Yaskawa INFORM job: X2_100(P)(125,-90).JBI

/JOB
//NAME X2_100(P)(125,-90)
//POS
///NPOS 573,573,573,27,0,0
///TOOL 0
///POSTYPE PULSE
///PULSE
C00000=3858,45070,-46943,-23358,97175,-79306
C00001=-126163,171030,121698,-25332,17066,-72423
///LIMIT ON
C00002=-15532,205449,169164,0,-1122,-37
C00003=-2035,205524,169313,0,-1142,-38
///LIMIT OFF
C00004=-24876,216658,221537,-34735,41227,28422
C00005=-32534,213651,221430,-43713,46730,30831
C00006=-90550,189136,203825,-30202,58765,18284
C00007=-119585,140470,218769,-27614,53519,-2911
C00008=-120519,138494,231532,-24554,52332,-6677
C00009=-121361,123084,224135,-22504,53325,-9347
C00010=-121726,115435,217146,-22627,53645,-9461
C00011=-121876,112275,214159,-22659,53833,-9521
C00012=-121870,108701,209945,-22450,54535,-9681
C00013=-121878,109205,210521,-22481,54446,-9661
C00014=-121910,109175,212145,-22779,53504,-9448
C00015=-121878,109205,210521,-22481,54446,-9661
C00016=-121362,120230,220888,-22358,53819,-9461
C00017=-121399,123144,224213,26030,40987,26163
C00018=-121766,115498,217228,25645,41349,26232
C00019=-121913,110359,211916,25262,41930,26397
C00020=-121910,108768,210034,25105,42240,26494
C00021=-121911,109318,210663,25153,42145,26465
C00022=-121945,109286,212284,25618,41227,26168
C00023=-121911,109318,210663,25153,42145,26465
C00024=-121395,120334,221016,25773,41460,26319
C00025=-121834,122785,223550,29969,46824,26161
C00026=-121859,115436,217233,29902,46923,26193
C00027=-121866,110818,212669,29698,47304,26325
C00028=-121863,108844,210335,29512,47673,26452
C00029=-121935,109447,211025,29521,47579,26410
C00030=-121969,109405,212635,29961,46698,26100
C00031=-121935,109447,211025,29521,47579,26410
C00032=-121897,120013,220389,29693,47285,26314
C00033=-121710,149750,244683,33916,46787,25442
C00034=-122130,167084,227684,35838,62010,28886
C00035=-121679,161325,224182,36290,61247,28722
C00036=-121494,157054,220841,36419,61089,28713
C00037=-121492,155796,219623,36386,61172,28744
C00038=-121498,156274,220057,36390,61156,28737
C00039=-121513,157313,222807,36761,60220,28378
C00040=-121498,156274,220057,36390,61156,28737
C00041=-122131,164491,225278,35793,62131,28930
C00042=-121153,166943,227356,19598,60055,30811
C00043=-121390,161131,223816,19656,59323,30620
C00044=-121486,157179,220857,19658,59138,30564
C00045=-121483,155572,219231,19626,59303,30596
C00046=-121495,156085,219721,19629,59269,30586
C00047=-121510,157133,222481,19854,58176,30378
C00048=-121495,156085,219721,19629,59269,30586
C00049=-121161,164380,224998,19569,60183,30833
C00050=-134270,166899,227330,-30052,67117,-21044
C00051=-134672,161022,223642,-30400,66383,-20931
C00052=-134827,157380,220874,-30511,66205,-20916
C00053=-134816,155436,218995,-30471,66344,-20953
C00054=-134842,155930,219452,-30490,66315,-20951
C00055=-135058,156963,222167,-30845,65285,-20702
C00056=-134842,155930,219452,-30490,66315,-20951
C00057=-134278,164319,224942,-30027,67241,-21080
C00058=-134522,188621,240209,-29351,55882,-39556
C00059=-134281,187845,227413,-27061,47780,-60505
C00060=-134637,183113,225522,-27632,46565,-60252
C00061=-134774,179835,223566,-27858,46107,-60152
C00062=-134763,178280,222255,-27854,46115,-60152
C00063=-134775,178711,222615,-27856,46112,-60156
C00064=-134965,180234,225747,-28400,45052,-59871
C00065=-134775,178711,222615,-27856,46112,-60156
C00066=-134277,185474,225522,-27083,47733,-60488
C00067=-128103,202093,243005,-900,47088,-2105
C00068=-121693,187846,227414,25459,51264,56132
C00069=-121495,183214,225706,25955,50017,55854
C00070=-121414,180043,223882,26152,49543,55743
C00071=-121411,178420,222512,26150,49549,55748
C00072=-121403,178860,222872,26150,49552,55751
C00073=-121416,180408,226053,26590,48508,55442
C00074=-121403,178860,222872,26150,49552,55751
C00075=-121682,185481,225516,25477,51219,56123
C00076=-121689,188183,227953,25513,51119,56094
C00077=-121490,183546,226247,26015,49869,55812
C00078=-121408,180079,224179,26215,49393,55704
C00079=-121407,178755,223064,26213,49397,55705
C00080=-121411,179182,223381,26203,49420,55711
C00081=-121423,180718,226547,26645,48380,55401
C00082=-121411,179182,223381,26203,49420,55711
C00083=-121690,185807,226020,25524,51091,56086
C00084=-123779,190470,236318,58172,45370,-30510
C00085=-122063,184657,229672,57761,45274,-29622
C00086=-121391,180820,225681,57548,45265,-29244
C00087=-121389,179381,224477,57547,45264,-29243
C00088=-121377,179861,224816,57519,45280,-29221
C00089=-121365,178277,221590,56564,45934,-28599
C00090=-121377,179861,224816,57519,45280,-29221
C00091=-121233,179889,223673,56966,45622,-28813
C00092=-120840,179898,223685,57074,45455,-28743
C00093=-121856,179870,223641,56791,45888,-28921
C00094=-124230,188212,233297,57460,45939,-30216
C00095=-135456,214682,237929,8760,44354,-9002
C00096=-135014,207234,230989,8630,44755,-8792
C00097=-134830,202547,226948,8592,44816,-8716
C00098=-134825,201671,226346,8603,44738,-8721
C00099=-134842,202253,226813,8604,44750,-8727
C00100=-134670,200231,223307,8417,45842,-8557
C00101=-134842,202253,226813,8604,44750,-8727
C00102=-135456,212819,236850,8805,44063,-9030
C00103=-144745,210021,243410,8185,41273,-14023
C00104=-162917,179999,233290,6575,38143,-23957
C00105=-161998,172707,226275,6517,38664,-23607
C00106=-162887,167099,219775,6342,39818,-23812
C00107=-162887,165781,218634,6340,39844,-23811
C00108=-162887,166055,218871,6340,39839,-23811
C00109=-162343,164612,215992,6206,40837,-23555
C00110=-162887,166055,218871,6340,39839,-23811
C00111=-162962,177992,231819,6593,38021,-23983
C00112=-147831,180663,236712,-46705,20975,10626
C00113=-148148,173122,227595,-43517,22125,9005
C00114=-148274,168937,222870,-42234,22650,8350
C00115=-148281,167110,221344,-42230,22650,8346
C00116=-148302,167857,221980,-42238,22637,8344
C00117=-147925,166248,218822,-40599,23599,7656
C00118=-148302,167857,221980,-42238,22637,8344
C00119=-147863,178628,235160,-46872,20902,10696
C00120=-134462,161839,227541,-33778,50638,-10353
C00121=-128292,130528,217892,-31335,63768,-21724
C00122=-129684,119449,220047,-34318,57761,-20007
C00123=-130320,112373,214177,-34735,57677,-20053
C00124=-130456,109465,211770,-34840,57652,-20062
C00125=-133214,109388,211257,-36497,57589,-20371
C00126=-136667,109271,210511,-38562,57521,-20784
C00127=-139224,109161,209855,-40060,57485,-21111
C00128=-138850,112080,212320,-39829,57519,-21074
C00129=-138002,119182,218308,-39302,57595,-20992
C00130=-116829,118715,218073,25020,47867,39145
C00131=-117081,112091,213071,24998,47591,39033
C00132=-116945,109370,210997,25124,47467,39017
C00133=-125403,109328,210939,20229,48081,38115
C00134=-125748,112035,212901,19975,48276,38114
C00135=-125224,118667,217955,20186,48522,38233
C00136=-124121,120753,219622,35413,60229,26204
C00137=-123486,114299,214861,35950,59841,26140
C00138=-122342,111487,212696,36731,59624,26198
C00139=-123646,102227,205116,46204,63991,23691
C00140=-125197,104926,207303,45145,64225,23601
C00141=-126541,111461,212474,44185,64527,23570
C00142=-123354,156374,234537,36141,60524,36841
C00143=-123006,163587,222304,33363,70023,40058
C00144=-122562,159556,221336,33872,68682,39742
C00145=-122328,157903,220938,34117,68123,39618
C00146=-120667,157882,220896,34940,67759,39903
C00147=-118950,157779,220838,35793,67346,40185
C00148=-123086,151768,218649,44650,69367,37665
C00149=-123645,153585,219325,44221,69895,37762
C00150=-124560,157673,220588,43425,71117,38069
C00151=-118179,162280,221931,19519,66647,42953
C00152=-118374,158121,220823,19639,65298,42675
C00153=-118267,155527,219476,19766,64809,42612
C00154=-124138,155466,219359,17061,65585,41471
C00155=-124017,158021,220644,17053,66071,41570
C00156=-123705,162202,221801,17023,67409,41838
C00157=-131226,163758,224551,-30632,74582,-25473
C00158=-131671,158900,222412,-31029,73469,-25265
C00159=-131767,156865,221384,-31140,73093,-25182
C00160=-137554,155593,218490,-34050,72807,-26431
C00161=-137282,157641,219617,-33852,73169,-26479
C00162=-136745,162505,221837,-33401,74244,-26683
C00163=-132458,177728,230704,-28826,51363,-58996
C00164=-131589,185090,225420,-26277,57937,-60697
C00165=-131989,181524,225146,-26843,56352,-60401
C00166=-132129,179690,224573,-27052,55792,-60292
C00167=-137018,178141,221655,-27936,55567,-61763
C00168=-136911,179846,222046,-27715,56157,-61897
C00169=-136440,196977,232068,-26852,58624,-62420
C00170=-123981,183157,222393,21512,66418,58052
C00171=-123825,180405,223212,21872,64600,57740
C00172=-123515,178835,223292,22117,63748,57656
C00173=-118554,178759,223273,23717,62772,58838
C00174=-118823,180539,223431,23475,63574,58935
C00175=-119074,183322,222662,23052,65379,59248
C00176=-122702,184077,222510,27150,66928,58165
C00177=-122303,181421,223407,27656,65122,57824
C00178=-121939,179837,223488,27962,64268,57706
C00179=-119147,179825,223466,28889,63614,58349
C00180=-122880,176137,223692,38896,64069,56161
C00181=-123433,177900,223899,38463,64850,56297
C00182=-124245,180658,223301,37680,66520,56676
C00183=-126373,202040,241637,26852,43466,21020
C00184=-128666,178893,235276,24840,16714,-14065
C00185=-128229,171381,226060,22241,18307,-12727
C00186=-128063,167759,221784,21279,19001,-12231
C00187=-126454,168065,222273,20329,18606,-11329
C00188=-113498,168020,221950,9782,17256,-2783
C00189=-116924,165235,218756,37372,21894,-17093
C00190=-117333,168644,222995,38850,21324,-17919
C00191=-117978,176136,232334,42331,20047,-19764
C00192=-122460,189534,236128,2418,24460,-9718
C00193=-126271,180528,223816,-31550,27550,-1309
C00194=-126367,172058,213874,-29849,29054,-2198
C00195=-127090,167664,208219,-28567,29945,-3048
C00196=-142506,160672,196064,-19689,30087,-11601
C00197=-142606,164949,201311,-20262,29094,-11331
C00198=-142831,174249,212461,-21540,27099,-10741
C00199=-90550,189136,203825,-30202,58765,18284
C00200=-32534,213651,221430,-43713,46730,30831
///LIMIT ON
C00201=-2035,205524,169313,0,-1142,-38
///LIMIT OFF
C00202=110357,194361,192639,11084,17793,24068
C00203=114624,170501,213981,27000,30394,20280
C00204=117760,152303,229663,38696,39653,17494
C00205=136745,136971,237540,47053,40245,16937
C00206=146994,113665,215692,48512,45897,19228
C00207=147943,109722,211385,48401,46737,19631
C00208=147915,107740,209041,48089,47029,19824
C00209=147921,108247,209621,48160,46963,19780
C00210=148534,108214,211137,49208,46239,19387
C00211=147921,108247,209621,48160,46963,19780
C00212=146752,119366,220398,48075,46495,19266
C00213=146769,122228,223642,-12245,42312,-23405
C00214=147600,114525,216379,-11673,42843,-23379
C00215=143912,110143,217361,-5106,40312,-21729
C00216=143912,106051,212649,-5023,41107,-21780
C00217=143912,106490,213159,-5032,41020,-21775
C00218=144459,106367,214517,-4806,40132,-21665
C00219=143912,108428,215397,-5071,40640,-21751
C00220=146723,119408,220432,-12150,42825,-23484
C00221=129935,127321,227469,-22947,42372,-25293
C00222=100595,140364,234928,-40781,43967,-29064
C00223=79895,121406,212050,-50395,45854,-33130
C00224=75281,118258,216394,-58069,38031,-30004
C00225=73869,113685,209088,-52247,40421,-30660
C00226=73869,110609,205591,-51722,40783,-30969
C00227=73869,110923,205950,-51776,40745,-30937
C00228=73085,111041,207234,-52885,40146,-30618
C00229=74213,115467,210577,-52057,40483,-30622
C00230=82018,121162,207620,-47441,48027,-34093
C00231=122098,148378,227955,-39779,54040,-25728
C00232=121690,165580,226205,-36203,61926,-29153
C00233=121256,163913,232537,-38022,57992,-27736
C00234=121056,160150,229731,-38195,57784,-27699
C00235=121055,158441,228110,-38151,57879,-27739
C00236=121062,158908,228526,-38154,57867,-27733
C00237=121061,159695,230985,-38583,56988,-27366
C00238=121062,158908,228526,-38154,57867,-27733
C00239=121746,167242,233775,-37439,58860,-27965
C00240=120722,169943,236314,-20799,56253,-30328
C00241=120960,164034,232760,-20897,55487,-30119
C00242=121057,160229,229930,-20909,55300,-30059
C00243=121055,158546,228333,-20881,55408,-30082
C00244=121067,159042,228799,-20882,55381,-30074
C00245=121067,159823,231250,-21156,54345,-29857
C00246=121067,159042,228799,-20882,55381,-30074
C00247=120732,167440,234058,-20772,56349,-30345
C00248=148415,169733,235789,37593,61151,22296
C00249=149007,163695,231894,38120,60456,22164
C00250=149231,159863,228946,38284,60282,22149
C00251=149211,158151,227325,38234,60380,22184
C00252=149239,158627,227750,38254,60361,22183
C00253=149676,159369,230053,38836,59445,21914
C00254=149239,158627,227750,38254,60361,22183
C00255=148408,167213,233502,37553,61243,22331
C00256=120948,174757,250553,37714,32624,49250
C00257=118901,165188,232218,31966,38533,51583
C00258=120946,159930,222884,30547,40745,53182
C00259=121038,156296,220141,30673,40571,53142
C00260=121036,154340,218237,30574,40715,53200
C00261=121048,154616,218515,30593,40687,53192
C00262=121049,155465,220596,31099,39958,52886
C00263=121048,154822,218707,30600,40677,53188
C00264=120729,163160,224069,29968,41598,53447
C00265=121377,165750,226457,-30289,41550,-53313
C00266=121143,159913,222862,-30795,40818,-53099
C00267=121047,156279,220118,-30922,40645,-53059
C00268=121045,154323,218215,-30823,40788,-53119
C00269=121036,154817,218686,-30845,40755,-53109
C00270=121036,155874,221461,-31554,39751,-52691
C00271=121036,154817,218686,-30845,40755,-53109
C00272=121366,163152,224045,-30207,41677,-53367
C00273=121272,196441,225736,-23884,56081,-57724
C00274=121089,199139,236729,-25537,51130,-56524
C00275=121004,196182,235381,-25789,50488,-56375
C00276=121002,194715,234291,-25819,50411,-56355
C00277=121006,195110,234541,-25802,50457,-56365
C00278=121007,196631,237575,-26196,49477,-56088
C00279=121006,195110,234541,-25802,50457,-56365
C00280=121299,201138,236064,-25032,52482,-56815
C00281=121488,201206,234672,-5139,48159,3169
C00282=137298,197580,228407,-4602,50872,8306
C00283=137722,195376,231059,-4778,48135,8578
C00284=139041,199622,244674,-11286,32429,11793
C00285=139041,197484,243237,-11354,32218,11828
C00286=139041,199622,244674,-11286,32429,11793
C00287=138787,198080,241716,-10937,33415,11530
C00288=139041,199622,244674,-11286,32429,11793
C00289=121299,208155,246357,-5458,44546,3313
C00290=123539,200771,239806,-5389,44887,4041
C00291=122594,197682,237757,-5423,44517,3747
C00292=122594,195371,236190,-5443,44297,3759
C00293=122594,197682,237757,-5423,44517,3747
C00294=122571,196051,234778,-5332,45507,3680
C00295=122594,197682,237757,-5423,44517,3747
C00296=121306,206138,245061,-5480,44308,3329
C00297=121658,212256,254439,-6066,40669,6202
C00298=109161,194767,243808,20461,40814,-3758
C00299=110406,186463,235065,20125,41665,-3120
C00300=110426,183388,231339,19860,42333,-2953
C00301=110426,181265,229707,19891,42253,-2973
C00302=110426,182012,230285,19880,42280,-2965
C00303=110530,180795,227899,19582,43058,-2746
C00304=110426,183866,231706,19851,42354,-2947
C00305=142983,174413,229445,40846,25339,-9857
C00306=144224,171221,225776,41394,24787,-9570
C00307=144224,167841,222912,41356,24808,-9552
C00308=144224,168628,223585,41369,24801,-9559
C00309=143936,167289,220827,40018,25660,-8977
C00310=142643,175710,231512,43415,24337,-11034
C00311=138046,186038,246419,52517,22458,-16631
C00312=135775,175505,231782,30106,22895,-7564
C00313=132887,170796,225962,29431,24495,-8118
C00314=133012,167528,222347,28819,24948,-7780
C00315=149327,160096,207563,18098,26717,2120
C00316=142622,177488,230472,24926,23040,-3139
C00317=137477,186722,245503,32144,20066,-8132
C00318=126529,166312,224180,-9540,26920,6556
C00319=130231,155715,216648,-10724,26396,8290
C00320=122698,152468,214837,12997,22490,-4012
C00321=121991,147575,209284,12791,23434,-4123
C00322=141345,142654,200759,11361,23339,4608
C00323=141508,151742,210671,11975,21923,4359
C00324=142241,168295,224091,-11275,28686,12573
C00325=118409,183246,223281,22704,61297,57282
C00326=118581,179790,223172,23116,59682,56982
C00327=119858,177440,221871,23553,59055,57217
C00328=122363,178731,225206,28497,55931,59046
C00329=123595,179764,223148,24469,58676,58234
C00330=123340,183247,223305,24003,60279,58531
C00331=123969,187046,227095,-21794,65540,-58072
C00332=123769,179484,222767,-22062,64364,-57894
C00333=124308,177722,222624,-22031,63705,-57614
C00334=119599,178184,223040,-23554,62794,-58733
C00335=118761,179531,222831,-23662,63378,-59098
C00336=119022,182337,222102,-23232,65173,-59409
C00337=122654,182929,221665,-27319,66777,-58337
C00338=122244,180255,222524,-27832,64982,-57999
C00339=122670,178331,221973,-27828,64506,-57752
C00340=119086,178516,222093,-29014,63676,-58577
C00341=121632,176313,222432,-35609,63813,-57115
C00342=123368,178358,224280,-38654,64701,-56471
C00343=124192,179556,222465,-37876,66329,-56835
C00344=123300,177441,230092,-34884,68799,-44911
C00345=123495,171160,238859,-36432,62561,-41346
C00346=123495,167355,235630,-36422,62587,-41356
C00347=124334,166434,238372,-37436,59393,-39895
C00348=118376,166713,238643,-40516,58128,-40736
C00349=118376,166713,238643,-40516,58128,-40736
C00350=120799,174385,242890,-38781,59689,-40830
C00351=118126,161343,221379,-19792,66498,-43092
C00352=118308,157164,220237,-19921,65161,-42814
C00353=119374,159410,226087,-20289,60239,-41711
C00354=124582,159325,225883,-17950,60958,-40729
C00355=124532,167340,231429,-17858,61624,-40849
C00356=143242,171476,234077,33692,69567,22108
C00357=145029,158578,222871,37922,70344,27214
C00358=146531,156505,221119,38712,69988,27450
C00359=149636,158546,225125,45286,65578,24312
C00360=145593,163818,228591,42995,67071,23935
C00361=129314,152311,241224,32836,60701,20495
C00362=134262,125348,219975,36015,59621,20953
C00363=136200,120757,215933,37173,59474,21178
C00364=138600,121552,220497,48290,55487,21652
C00365=129739,126079,224796,42731,56443,20863
C00366=123968,133718,232687,39402,56414,20088
C00367=116671,118195,219736,-25901,46707,-38928
C00368=118115,111302,212748,-24760,47506,-38978
C00369=118703,106589,208138,-24267,47934,-39019
C00370=126682,106493,207892,-19649,48585,-38165
C00371=117444,111276,212730,-25153,47452,-39048
C00372=124109,119988,219209,-35802,60097,-26259
C00373=123452,113507,214395,-36349,59725,-26200
C00374=123794,109050,210148,-36021,60020,-26273
C00375=117612,109054,210103,-40010,59333,-26782
C00376=118160,111552,216388,-45062,55465,-25714
C00377=121329,120470,223550,-42877,55942,-25575
C00378=129083,121917,227984,-46752,58292,-19813
C00379=114229,133215,224760,-34569,55636,-15897
C00380=115215,137513,213650,-31198,63454,-18326
C00381=115698,129470,194907,-29425,69976,-20075
C00382=106762,152299,200628,-28970,57173,-24551
C00383=106762,152299,184780,-28970,-3668,-24551
C00384=106762,172700,182835,-23749,-4416,-26879
C00385=106762,173596,155880,-23749,-4416,-26879
C00386=27327,173596,155880,-23749,-4416,-26879
C00387=61821,209309,227101,13653,32656,17858
C00388=117760,152303,229663,38696,39653,17494
C00389=136745,136971,237540,47053,40245,16937
C00390=146994,113665,215692,48512,45897,19228
C00391=147943,109722,211385,48401,46737,19631
C00392=147915,107740,209041,48089,47029,19824
C00393=147921,108247,209621,48160,46963,19780
C00394=148534,108214,211137,49208,46239,19387
C00395=147921,108247,209621,48160,46963,19780
C00396=146752,119366,220398,48075,46495,19266
C00397=146769,122228,223642,-12245,42312,-23405
C00398=147600,114525,216379,-11673,42843,-23379
C00399=150410,110151,217690,-10757,39930,-22674
C00400=147891,107738,209025,-11299,43871,-23478
C00401=153573,108674,222079,-9620,36586,-21959
C00402=148504,108258,211178,-11182,42854,-23269
C00403=153573,108674,222079,-9620,36586,-21959
C00404=146723,119408,220432,-12150,42825,-23484
C00405=129935,127321,227469,-22947,42372,-25293
C00406=100595,140364,234928,-40781,43967,-29064
C00407=81913,119649,206036,-47366,48141,-34193
C00408=81142,111914,198932,-47506,48252,-34466
C00409=80567,105530,192695,-47437,48513,-34785
C00410=80567,103424,190213,-47154,48820,-34981
C00411=79896,104610,192938,-48190,47941,-34592
C00412=79367,104896,194278,-48926,47369,-34348
C00413=81288,108115,194243,-46832,48931,-34860
C00414=82018,116513,202458,-46931,48572,-34441
C00415=122104,148543,228477,-39885,53858,-25643
C00416=121690,165580,226205,-36203,61926,-29153
C00417=121228,159785,222619,-36652,61188,-29000
C00418=121039,155988,219702,-36787,61016,-28984
C00419=121038,154211,217971,-36739,61139,-29031
C00420=121044,154693,218413,-36744,61121,-29023
C00421=121043,155760,221200,-37127,60178,-28661
C00422=121044,154693,218413,-36744,61121,-29023
C00423=121694,162967,223761,-36153,62058,-29201
C00424=120722,165761,226456,-19970,59936,-31049
C00425=120948,159926,222866,-20032,59223,-30862
C00426=121040,156088,219926,-20029,59083,-30814
C00427=121038,154338,218222,-19999,59222,-30841
C00428=121049,154854,218719,-20002,59186,-30831
C00429=121049,155913,221496,-20240,58090,-30621
C00430=121049,154854,218719,-20002,59186,-30831
C00431=120732,163185,224070,-19939,60073,-31072
C00432=147021,165785,226508,35831,64459,23179
C00433=147568,159794,222565,36267,63796,23080
C00434=147776,155921,219507,36395,63658,23083
C00435=147758,154144,217781,36345,63784,23124
C00436=147784,154635,218233,36365,63757,23122
C00437=148179,155632,220846,36870,62776,22859
C00438=147784,154635,218233,36365,63757,23122
C00439=147016,163193,224095,35787,64586,23223
C00440=120935,171934,242189,34504,35645,50983
C00441=120720,165768,226479,30046,41476,53396
C00442=120946,159930,222884,30547,40745,53182
C00443=121038,156296,220141,30673,40571,53142
C00444=121036,154340,218237,30574,40715,53200
C00445=121048,154616,218515,30593,40687,53192
C00446=121049,155465,220596,31099,39958,52886
C00447=121048,154822,218707,30600,40677,53188
C00448=120729,163160,224069,29968,41598,53447
C00449=121377,165750,226457,-30289,41550,-53313
C00450=121143,159913,222862,-30795,40818,-53099
C00451=121047,156279,220118,-30922,40645,-53059
C00452=121045,154323,218215,-30823,40788,-53119
C00453=121036,154817,218686,-30845,40755,-53109
C00454=121036,155874,221461,-31554,39751,-52691
C00455=121036,154817,218686,-30845,40755,-53109
C00456=121366,163152,224045,-30207,41677,-53367
C00457=121272,196441,225736,-23884,56081,-57724
C00458=121073,192434,224897,-24336,54621,-57437
C00459=120992,189535,223518,-24533,54018,-57314
C00460=120990,188039,222350,-24548,53971,-57303
C00461=120994,188436,222615,-24536,54010,-57311
C00462=120994,190244,226010,-24889,52951,-57041
C00463=120994,188436,222615,-24536,54010,-57311
C00464=121274,194182,224023,-23912,55983,-57699
C00465=121488,201206,234672,-5139,48159,3169
C00466=137298,197580,228407,-4602,50872,8306
C00467=137298,191509,224279,-4639,50294,8333
C00468=139269,198483,245774,-16664,26320,14172
C00469=139269,196637,244517,-16766,26152,14223
C00470=139269,198483,245774,-16664,26320,14172
C00471=139075,197379,243601,-16166,27033,13866
C00472=139269,198483,245774,-16664,26320,14172
C00473=121273,201949,235341,-5146,48120,3100
C00474=123414,194344,228329,-5073,48626,3789
C00475=122511,191235,226161,-5095,48321,3503
C00476=122511,188904,224500,-5108,48148,3511
C00477=122511,191235,226161,-5095,48321,3503
C00478=122490,189334,222835,-5015,49386,3440
C00479=122511,191235,226161,-5095,48321,3503
C00480=121280,199935,233985,-5161,47920,3112
C00481=121614,206656,244155,-5683,44100,5953
C00482=121602,191150,235422,-5966,40449,9428
C00483=121174,183490,227904,-5875,41115,9232
C00484=121005,180342,224725,-5833,41444,9150
C00485=121003,177643,222663,-5847,41326,9158
C00486=121008,178404,223350,-5851,41294,9161
C00487=121008,176471,219820,-5719,42467,9082
C00488=121008,178404,223350,-5851,41294,9161
C00489=121606,189290,234231,-5993,40228,9445
C00490=147345,179625,236056,47140,21312,-11138
C00491=147690,172068,226895,43950,22458,-9504
C00492=147826,168050,222291,42659,22984,-8839
C00493=147834,166033,220594,42645,22988,-8830
C00494=147855,166783,221239,42657,22973,-8830
C00495=147492,165159,218049,41004,23935,-8131
C00496=147855,166783,221239,42657,22973,-8830
C00497=147377,177583,234490,47295,21243,-11203
C00498=135775,175505,231782,30106,22895,-7564
C00499=139825,168083,220832,25470,24638,-4146
C00500=139700,165046,217320,24964,25206,-3934
C00501=152174,156983,201769,15688,28186,4094
C00502=150364,166319,215167,18488,25143,2197
C00503=147525,184400,240334,25395,19839,-1947
C00504=126529,166312,224180,-9540,26920,6556
C00505=130231,155715,216648,-10724,26396,8290
C00506=130045,149819,208548,-10003,28305,7869
C00507=131869,147843,216891,-25172,12050,11560
C00508=149055,140634,197724,-21214,26307,18683
C00509=148313,150562,204331,-12308,32779,14754
C00510=148313,166205,218654,-12570,32021,14892
C00511=118409,183246,223281,22704,61297,57282
C00512=118581,179790,223172,23116,59682,56982
C00513=119613,177433,221860,23486,59108,57157
C00514=124091,177390,221715,24682,58266,58283
C00515=123595,179764,223148,24469,58676,58234
C00516=123340,183247,223305,24003,60279,58531
C00517=123938,190075,227776,-21625,66593,-58285
C00518=123769,179484,222767,-22062,64364,-57894
C00519=123980,177747,222673,-22141,63629,-57689
C00520=118975,177987,223072,-23779,62559,-58856
C00521=118761,179531,222831,-23662,63378,-59098
C00522=119022,182337,222102,-23232,65173,-59409
C00523=122654,182929,221665,-27319,66777,-58337
C00524=122244,180255,222524,-27832,64982,-57999
C00525=122348,178243,222080,-27959,64333,-57799
C00526=119084,177910,221892,-29058,63509,-58532
C00527=123183,174594,222305,-38836,64062,-56290
C00528=123368,176775,223017,-38664,64673,-56460
C00529=124192,179556,222465,-37876,66329,-56835
C00530=123300,177441,230092,-34884,68799,-44911
C00531=122965,162591,221617,-33646,69855,-40187
C00532=122509,158537,220602,-34164,68528,-39873
C00533=122656,156640,219931,-34208,68093,-39694
C00534=118888,156854,220084,-36079,67235,-40332
C00535=123197,150890,218022,-44883,69229,-37756
C00536=123579,152565,218570,-44547,69710,-37880
C00537=124509,156681,219892,-43743,70915,-38181
C00538=118126,161343,221379,-19792,66498,-43092
C00539=118308,157164,220237,-19921,65161,-42814
C00540=119071,154535,218903,-19652,64761,-42579
C00541=124368,154518,218802,-17210,65477,-41554
C00542=123968,157132,220198,-17330,65894,-41703
C00543=123666,161333,221389,-17292,67221,-41971
C00544=144355,163571,225284,37353,71372,27423
C00545=145029,158578,222871,37922,70344,27214
C00546=146175,156230,221157,38559,69945,27345
C00547=151129,153949,216102,40712,70190,28712
C00548=150395,156248,217650,40288,70560,28668
C00549=149652,161243,220185,39700,71542,28858
C00550=132795,148549,237387,35039,60818,21489
C00551=129694,120788,221943,34103,57517,19821
C00552=131382,111553,213551,35044,57698,20084
C00553=143552,107861,207554,42137,57676,21682
C00554=150345,107155,204350,45732,57861,22855
C00555=138916,111308,211941,39557,57554,20977
C00556=138073,118434,217968,39036,57618,20892
C00557=116671,118195,219736,-25901,46707,-38928
C00558=118115,111302,212748,-24760,47506,-38978
C00559=118365,108555,210469,-24620,47519,-38949
C00560=126723,108483,210190,-19740,48219,-38083
C00561=125733,111262,212625,-20332,48091,-38177
C00562=125221,117920,217723,-20539,48325,-38292
C00563=124109,119988,219209,-35802,60097,-26259
C00564=123452,113507,214395,-36349,59725,-26200
C00565=123456,109791,211594,-36410,59571,-26144
C00566=117908,109386,211182,-40002,58985,-26593
C00567=124626,100214,203389,-45889,64097,-23721
C00568=125145,104077,206766,-45571,64098,-23654
C00569=126515,110647,212006,-44599,64385,-23614
C00570=114229,133215,224760,-34569,55636,-15897
C00571=58944,196489,225704,17941,27585,14980
C00572=-5072,204191,177105,2520,2910,2072
BC00000=46343,515539,1075137
BC00001=134211,257442,1075137
BC00002=1577,514581,1075193
///LIMIT ON
BC00003=1577,-59411,1075193
BC00004=21651,-83121,1075193
BC00005=24420,-86391,1075193
BC00006=182796,-159531,881707
BC00007=261191,-81513,996983
BC00008=265032,-63260,961437
BC00009=267226,-52830,941125
BC00010=267226,-52830,941125
BC00011=267226,-52830,941125
BC00012=267226,-52830,941125
BC00013=267226,-52830,941125
BC00014=267226,-52830,941125
BC00015=267226,-52830,941125
BC00016=267226,-52830,941125
BC00017=280671,-69653,979309
BC00018=280671,-69653,979309
BC00019=280671,-69653,979309
BC00020=280671,-69653,979309
BC00021=280671,-69653,979309
BC00022=280671,-69653,979309
BC00023=280671,-69653,979309
BC00024=280671,-69653,979309
BC00025=340059,-63189,958778
BC00026=340059,-63189,958778
BC00027=340059,-63189,958778
BC00028=340059,-63189,958778
BC00029=340059,-63189,958778
BC00030=340059,-63189,958778
BC00031=340059,-63189,958778
BC00032=340059,-63189,958778
BC00033=335398,-76723,919166
BC00034=322582,-113941,810232
BC00035=322582,-113941,810232
BC00036=322582,-113941,810232
BC00037=322582,-113941,810232
BC00038=322582,-113941,810232
BC00039=322582,-113941,810232
BC00040=322582,-113941,810232
BC00041=322582,-113941,810232
BC00042=280667,-107560,836160
BC00043=280667,-107560,836160
BC00044=280667,-107560,836160
BC00045=280667,-107560,836160
BC00046=280667,-107560,836160
BC00047=280667,-107560,836160
BC00048=280667,-107560,836160
BC00049=280667,-107560,836160
BC00050=310567,-93619,803899
BC00051=310567,-93619,803899
BC00052=310567,-93619,803899
BC00053=310567,-93619,803899
BC00054=310567,-93619,803899
BC00055=310567,-93619,803899
BC00056=310567,-93619,803899
BC00057=310567,-93619,803899
BC00058=310965,-106510,799405
BC00059=311390,-120260,794612
BC00060=311390,-120260,794612
BC00061=311390,-120260,794612
BC00062=311390,-120260,794612
BC00063=311390,-120260,794612
BC00064=311390,-120260,794612
BC00065=311390,-120260,794612
BC00066=311390,-120260,794612
BC00067=292086,-121797,794251
BC00068=272781,-123335,793890
BC00069=272781,-123335,793890
BC00070=272781,-123335,793889
BC00071=272781,-123335,793890
BC00072=272781,-123335,793890
BC00073=272781,-123335,793890
BC00074=272781,-123335,793890
BC00075=272781,-123335,793890
BC00076=341329,-123426,794084
BC00077=341329,-123426,794084
BC00078=341329,-123426,794084
BC00079=341329,-123426,794084
BC00080=341329,-123426,794084
BC00081=341329,-123426,794084
BC00082=341329,-123426,794084
BC00083=341329,-123426,794084
BC00084=311173,-145946,723752
BC00085=311173,-145946,723752
BC00086=311173,-145946,723752
BC00087=311173,-145946,723752
BC00088=311173,-145946,723752
BC00089=311173,-145946,723752
BC00090=311173,-145946,723752
BC00091=311173,-145946,723752
BC00092=311173,-145946,723752
BC00093=311173,-145946,723752
BC00094=311173,-145946,723752
BC00095=368417,-159833,659013
BC00096=368417,-159833,659013
BC00097=368417,-159833,659013
BC00098=368417,-159833,659013
BC00099=368417,-159833,659013
BC00100=368417,-159833,659013
BC00101=368417,-159833,659013
BC00102=368417,-159833,659013
BC00103=371175,-130977,746316
BC00104=376801,-72111,924416
BC00105=376801,-72111,924416
BC00106=376801,-72111,924416
BC00107=376801,-72111,924416
BC00108=376801,-72111,924416
BC00109=376801,-72111,924414
BC00110=376801,-72111,924416
BC00111=376801,-72111,924416
BC00112=341502,-110623,881707
BC00113=341502,-110623,881707
BC00114=341502,-110623,881707
BC00115=341502,-110623,881707
BC00116=341502,-110623,881707
BC00117=341502,-110623,881707
BC00118=341502,-110623,881707
BC00119=341502,-110623,881707
BC00120=317229,-102231,901443
BC00121=301231,-72103,952987
BC00122=300570,-48582,912240
BC00123=300570,-48582,912240
BC00124=300570,-48582,912238
BC00125=300570,-48582,912240
BC00126=300570,-48582,912240
BC00127=300570,-48582,912240
BC00128=300570,-48582,912240
BC00129=300570,-48582,912240
BC00130=280392,-58723,951442
BC00131=280392,-58723,951442
BC00132=280392,-58723,951442
BC00133=280392,-58723,951442
BC00134=280392,-58723,951442
BC00135=280392,-58723,951442
BC00136=316381,-56573,892692
BC00137=316381,-56573,892692
BC00138=316381,-56573,892692
BC00139=316381,-56573,892692
BC00140=316381,-56573,892692
BC00141=316381,-56573,892692
BC00142=316378,-102850,892874
BC00143=316296,-103943,772800
BC00144=316296,-103943,772800
BC00145=316296,-103943,772800
BC00146=316296,-103943,772800
BC00147=316296,-103943,772800
BC00148=316296,-103943,772800
BC00149=316296,-103943,772800
BC00150=316296,-103943,772800
BC00151=280455,-96630,809993
BC00152=280455,-96630,809993
BC00153=280455,-96630,809993
BC00154=280455,-96630,809993
BC00155=280455,-96630,809993
BC00156=280455,-96630,809993
BC00157=313485,-85360,768647
BC00158=313485,-85360,768647
BC00159=313485,-85360,768647
BC00160=313485,-85360,768647
BC00161=313485,-85360,768647
BC00162=313485,-85360,768647
BC00163=312825,-103474,920081
BC00164=312211,-104211,778577
BC00165=312211,-104211,778577
BC00166=312212,-104211,778575
BC00167=312212,-104211,778575
BC00168=312211,-104211,778577
BC00169=312211,-104211,778577
BC00170=271148,-98769,766614
BC00171=271148,-98769,766614
BC00172=271148,-98769,766614
BC00173=271148,-98769,766614
BC00174=271148,-98769,766614
BC00175=271148,-98769,766614
BC00176=325606,-102154,751502
BC00177=325606,-102154,751502
BC00178=325606,-102154,751502
BC00179=325606,-102154,751502
BC00180=325606,-102154,751502
BC00181=325606,-102154,751502
BC00182=325606,-102154,751502
BC00183=333034,-134164,767871
BC00184=339129,-149656,848222
BC00185=339129,-149656,848222
BC00186=339128,-149655,848221
BC00187=339129,-149656,848222
BC00188=339129,-149656,848222
BC00189=339129,-149656,848222
BC00190=339129,-149656,848222
BC00191=339129,-149656,848222
BC00192=327972,-150195,844855
BC00193=317352,-148908,839217
BC00194=317352,-148908,839217
BC00195=317352,-148908,839217
BC00196=317352,-148908,839217
BC00197=317352,-148908,839217
BC00198=317352,-148908,839217
BC00199=182796,-159531,881707
BC00200=24420,-86391,1075193
BC00201=1577,-59411,1075193
///LIMIT OFF
BC00202=66886,568997,1042628
BC00203=92444,428784,1010343
BC00204=92897,349346,986620
BC00205=134271,323227,963040
BC00206=152063,311995,952900
BC00207=153659,310988,951990
BC00208=153659,310988,951990
BC00209=153659,310988,951990
BC00210=153659,310988,951990
BC00211=153659,310988,951990
BC00212=153659,310988,951990
BC00213=157626,318421,980677
BC00214=157626,318421,980677
BC00215=157626,306857,980677
BC00216=157626,306857,980677
BC00217=157626,306857,980677
BC00218=157626,306857,980677
BC00219=157626,306857,980677
BC00220=157626,318421,980677
BC00221=135895,324391,972471
BC00222=98646,334624,958405
BC00223=86230,316808,953716
BC00224=86230,311202,953716
BC00225=86230,311202,953716
BC00226=86230,311202,953716
BC00227=86230,311202,953716
BC00228=86230,311202,953716
BC00229=86230,311202,953716
BC00230=86230,325332,953716
BC00231=152073,357351,961616
BC00232=152073,370738,812197
BC00233=152073,359985,812197
BC00234=152073,359985,812197
BC00235=152073,359985,812197
BC00236=152073,359985,812197
BC00237=152073,359985,812197
BC00238=152073,359985,812197
BC00239=152073,359985,812197
BC00240=110057,353717,838001
BC00241=110057,353717,838001
BC00242=110057,353717,838001
BC00243=110057,353717,838001
BC00244=110057,353717,838001
BC00245=110057,353717,838001
BC00246=110057,353717,838001
BC00247=110057,353717,838001
BC00248=175407,329283,804361
BC00249=175407,329283,804361
BC00250=175407,329283,804361
BC00251=175407,329283,804361
BC00252=175407,329283,804361
BC00253=175407,329283,804361
BC00254=175407,329283,804361
BC00255=175407,329283,804361
BC00256=99689,342192,928572
BC00257=99689,342192,928572
BC00258=99689,352945,928572
BC00259=99689,352945,928572
BC00260=99689,352945,928572
BC00261=99689,352945,928572
BC00262=99690,352945,928571
BC00263=99689,352945,928572
BC00264=99689,352945,928572
BC00265=102794,353410,929381
BC00266=102794,353410,929381
BC00267=102794,353410,929381
BC00268=102794,353410,929381
BC00269=102794,353410,929381
BC00270=102794,353410,929381
BC00271=102794,353410,929381
BC00272=102794,353410,929381
BC00273=171341,390855,723900
BC00274=171341,380102,723900
BC00275=171341,380102,723900
BC00276=171341,380102,723900
BC00277=171341,380102,723900
BC00278=171341,380102,723900
BC00279=171341,380102,723900
BC00280=171341,380102,723900
BC00281=152795,392127,745599
BC00282=152795,392127,745599
BC00283=152795,385982,745599
BC00284=152795,385982,745599
BC00285=152795,385982,745599
BC00286=152795,385982,745599
BC00287=152795,385982,745599
BC00288=152795,385982,745599
BC00289=152795,381374,745599
BC00290=152795,381374,745599
BC00291=152795,381372,745596
BC00292=152795,381372,745596
BC00293=152795,381372,745596
BC00294=152795,381372,745596
BC00295=152795,381372,745596
BC00296=152795,381374,745599
BC00297=127624,372344,791394
BC00298=96392,361311,848216
BC00299=96392,361311,848216
BC00300=96392,361311,848216
BC00301=96392,361311,848216
BC00302=96392,361311,848216
BC00303=96392,361311,848216
BC00304=96392,361311,848216
BC00305=166858,366831,881738
BC00306=168143,366933,882362
BC00307=168143,366933,882362
BC00308=168143,366933,882362
BC00309=168143,366933,882362
BC00310=168143,366933,882362
BC00311=169598,367048,883068
BC00312=170817,374740,895100
BC00313=170820,374784,895167
BC00314=170820,374784,895167
BC00315=170829,374911,895362
BC00316=170829,374911,895362
BC00317=170831,374937,895402
BC00318=174622,382655,949814
BC00319=174622,382655,949814
BC00320=174623,382651,949823
BC00321=174623,382651,949823
BC00322=174665,382529,950104
BC00323=174665,382529,950104
BC00324=174666,382524,950113
BC00325=101409,363347,778304
BC00326=101409,363347,778304
BC00327=101409,363348,778302
BC00328=101409,363347,778303
BC00329=101409,363347,778304
BC00330=101409,363347,778304
BC00331=115011,355192,768709
BC00332=101979,355192,768709
BC00333=101979,355192,768709
BC00334=101979,355192,768709
BC00335=101979,355192,768709
BC00336=101979,355192,768709
BC00337=156450,358059,753624
BC00338=156450,358059,753624
BC00339=156450,358059,753624
BC00340=156450,358059,753624
BC00341=156450,358059,753624
BC00342=156450,358059,753624
BC00343=156450,358059,753624
BC00344=148838,358978,771431
BC00345=148358,349966,772279
BC00346=148358,349966,772279
BC00347=148358,349966,772279
BC00348=148358,349966,772279
BC00349=148358,349966,772279
BC00350=148358,349966,772279
BC00351=111086,353070,811970
BC00352=111086,353070,811970
BC00353=111086,353070,811970
BC00354=111086,353070,811970
BC00355=111086,353070,811970
BC00356=174257,332985,770647
BC00357=179294,331383,767352
BC00358=179294,331383,767352
BC00359=179294,331383,767352
BC00360=179294,331383,767352
BC00361=141072,318668,849125
BC00362=140860,318424,871943
BC00363=140860,318424,871943
BC00364=140860,318424,871943
BC00365=140860,318424,871943
BC00366=140860,318424,871943
BC00367=111313,315083,952947
BC00368=111313,315083,952947
BC00369=111313,315083,952947
BC00370=111313,315083,952947
BC00371=111313,315083,952947
BC00372=147008,312571,894102
BC00373=147008,312571,894102
BC00374=147008,312571,894102
BC00375=147008,312571,894102
BC00376=147008,312571,894102
BC00377=147008,312571,894102
BC00378=147008,312571,894102
BC00379=115348,333024,923162
BC00380=115348,333024,923162
BC00381=115349,359008,1050367
BC00382=115349,380944,1050367
BC00383=115349,443750,1050367
BC00384=115349,500340,1050367
BC00385=115349,585882,1050367
BC00386=11136,585882,1050367
BC00387=140184,427082,1056800
BC00388=263325,349346,986620
BC00389=304699,323227,963040
BC00390=322491,311995,952900
BC00391=324087,310988,951990
BC00392=324087,310988,951990
BC00393=324087,310988,951990
BC00394=324087,310988,951990
BC00395=324087,310988,951990
BC00396=324087,310988,951990
BC00397=328054,318421,980677
BC00398=328054,318421,980677
BC00399=328054,306857,980677
BC00400=328054,318421,980677
BC00401=328054,294465,980677
BC00402=328054,318421,980677
BC00403=328054,294465,980677
BC00404=328054,318421,980677
BC00405=306323,324391,972471
BC00406=269074,334624,958405
BC00407=256658,325332,953716
BC00408=256658,325332,953716
BC00409=256658,325332,953716
BC00410=256658,325332,953716
BC00411=256658,322580,953716
BC00412=256658,322580,953716
BC00413=256658,325332,953716
BC00414=256658,325332,953716
BC00415=322501,370738,961616
BC00416=322501,370738,812197
BC00417=322501,370738,812197
BC00418=322501,370738,812197
BC00419=322501,370738,812197
BC00420=322501,370738,812197
BC00421=322501,370738,812197
BC00422=322501,370738,812197
BC00423=322501,370738,812197
BC00424=280485,364470,838001
BC00425=280485,364470,838001
BC00426=280485,364470,838001
BC00427=280485,364470,838001
BC00428=280485,364470,838001
BC00429=280485,364470,838001
BC00430=280485,364470,838001
BC00431=280485,364470,838001
BC00432=345835,340036,804361
BC00433=345835,340036,804361
BC00434=345835,340036,804361
BC00435=345835,340036,804361
BC00436=345835,340036,804361
BC00437=345835,340036,804361
BC00438=345835,340036,804361
BC00439=345835,340036,804361
BC00440=270117,352945,928572
BC00441=270117,352945,928572
BC00442=270117,352945,928572
BC00443=270117,352945,928572
BC00444=270117,352945,928572
BC00445=270117,352945,928572
BC00446=270118,352945,928571
BC00447=270117,352945,928572
BC00448=270117,352945,928572
BC00449=273222,353410,929381
BC00450=273222,353410,929381
BC00451=273222,353410,929381
BC00452=273222,353410,929381
BC00453=273222,353410,929381
BC00454=273222,353410,929381
BC00455=273222,353410,929381
BC00456=273222,353410,929381
BC00457=341769,390855,723900
BC00458=341769,390855,723900
BC00459=341769,390855,723900
BC00460=341769,390855,723900
BC00461=341769,390855,723900
BC00462=341769,390855,723900
BC00463=341769,390855,723900
BC00464=341769,390855,723900
BC00465=323223,392127,745599
BC00466=323223,392127,745599
BC00467=323223,392127,745599
BC00468=323223,392127,745599
BC00469=323223,392127,745599
BC00470=323223,392127,745599
BC00471=323223,392127,745599
BC00472=323223,392127,745599
BC00473=323223,392127,745599
BC00474=323223,392127,745599
BC00475=323223,392125,745596
BC00476=323223,392125,745596
BC00477=323223,392125,745596
BC00478=323223,392125,745596
BC00479=323223,392125,745596
BC00480=323223,392127,745599
BC00481=298052,383097,791394
BC00482=262282,370265,856472
BC00483=262282,370265,856472
BC00484=262282,370265,856472
BC00485=262282,370265,856472
BC00486=262282,370265,856472
BC00487=262282,370265,856472
BC00488=262282,370265,856472
BC00489=262282,370265,856472
BC00490=340700,367102,883396
BC00491=340700,367102,883396
BC00492=340700,367102,883396
BC00493=340700,367102,883396
BC00494=340700,367102,883396
BC00495=340700,367102,883396
BC00496=340700,367102,883396
BC00497=340700,367102,883396
BC00498=341245,374740,895100
BC00499=341248,374789,895175
BC00500=341248,374789,895175
BC00501=341259,374937,895402
BC00502=341259,374937,895402
BC00503=341259,374937,895402
BC00504=345050,382655,949814
BC00505=345050,382655,949814
BC00506=345050,382655,949814
BC00507=345055,382639,949850
BC00508=345094,382524,950114
BC00509=345094,382524,950114
BC00510=345094,382524,950114
BC00511=271837,363347,778304
BC00512=271837,363347,778304
BC00513=271837,363348,778302
BC00514=271837,363347,778303
BC00515=271837,363347,778304
BC00516=271837,363347,778304
BC00517=272407,355192,768709
BC00518=272407,355192,768709
BC00519=272407,355192,768709
BC00520=272407,355192,768709
BC00521=272407,355192,768709
BC00522=272407,355192,768709
BC00523=326878,358059,753624
BC00524=326878,358059,753624
BC00525=326878,358059,753624
BC00526=326878,358059,753624
BC00527=326878,358059,753624
BC00528=326878,358059,753624
BC00529=326878,358059,753624
BC00530=319266,358978,771431
BC00531=317411,360013,774707
BC00532=317411,360013,774707
BC00533=317411,360013,774707
BC00534=317411,360013,774707
BC00535=317411,360013,774707
BC00536=317411,360013,774707
BC00537=317411,360013,774707
BC00538=281514,353070,811970
BC00539=281514,353070,811970
BC00540=281514,353070,811970
BC00541=281514,353070,811970
BC00542=281514,353070,811970
BC00543=281514,353070,811970
BC00544=349722,331383,767352
BC00545=349722,331383,767352
BC00546=349722,331383,767352
BC00547=349722,331383,767352
BC00548=349722,331383,767352
BC00549=349722,331383,767352
BC00550=305745,317122,860141
BC00551=301321,303767,911398
BC00552=301321,303767,911398
BC00553=322076,303767,911398
BC00554=322076,303767,911398
BC00555=301321,303767,911398
BC00556=301321,303767,911398
BC00557=281741,315083,952947
BC00558=281741,315083,952947
BC00559=281741,315083,952947
BC00560=281741,315083,952947
BC00561=281741,315083,952947
BC00562=281741,315083,952947
BC00563=317436,312571,894102
BC00564=317436,312571,894102
BC00565=317436,312571,894102
BC00566=317436,312571,894102
BC00567=317436,312571,894102
BC00568=317436,312571,894102
BC00569=317436,312571,894102
BC00570=285776,333024,923162
BC00571=140184,427082,1056800
BC00572=21044,502292,1072610
EC00000=-1108551,372643
EC00001=-1108551,372643
EC00002=-1108551,372643
EC00003=-1108551,372643
EC00004=-1108551,372643
EC00005=-1108551,372643
EC00006=-1108551,372643
EC00007=-1108551,372643
EC00008=-1108551,372643
EC00009=-1108551,372643
EC00010=-1108551,372643
EC00011=-1108551,372643
EC00012=-1108551,372643
EC00013=-1108551,372643
EC00014=-1108551,372643
EC00015=-1108551,372643
EC00016=-1108551,372643
EC00017=-1108551,372643
EC00018=-1108551,372643
EC00019=-1108551,372643
EC00020=-1108551,372643
EC00021=-1108551,372643
EC00022=-1108551,372643
EC00023=-1108551,372643
EC00024=-1108551,372643
EC00025=-1108551,372643
EC00026=-1108551,372643
EC00027=-1108551,372643
EC00028=-1108551,372643
EC00029=-1108551,372643
EC00030=-1108551,372643
EC00031=-1108551,372643
EC00032=-1108551,372643
EC00033=-1108551,372643
EC00034=-1108551,372643
EC00035=-1108551,372643
EC00036=-1108551,372643
EC00037=-1108551,372643
EC00038=-1108551,372643
EC00039=-1108551,372643
EC00040=-1108551,372643
EC00041=-1108551,372643
EC00042=-1108551,372643
EC00043=-1108551,372643
EC00044=-1108551,372643
EC00045=-1108551,372643
EC00046=-1108551,372643
EC00047=-1108551,372643
EC00048=-1108551,372643
EC00049=-1108551,372643
EC00050=-1108551,372643
EC00051=-1108551,372643
EC00052=-1108551,372643
EC00053=-1108551,372643
EC00054=-1108551,372643
EC00055=-1108551,372643
EC00056=-1108551,372643
EC00057=-1108551,372643
EC00058=-1108551,372643
EC00059=-1108551,372643
EC00060=-1108551,372643
EC00061=-1108551,372643
EC00062=-1108551,372643
EC00063=-1108551,372643
EC00064=-1108551,372643
EC00065=-1108551,372643
EC00066=-1108551,372643
EC00067=-1108551,372643
EC00068=-1108551,372643
EC00069=-1108551,372643
EC00070=-1108550,372643
EC00071=-1108551,372643
EC00072=-1108551,372643
EC00073=-1108551,372643
EC00074=-1108551,372643
EC00075=-1108551,372643
EC00076=-1108551,372643
EC00077=-1108551,372643
EC00078=-1108551,372643
EC00079=-1108551,372643
EC00080=-1108551,372643
EC00081=-1108551,372643
EC00082=-1108551,372643
EC00083=-1108551,372643
EC00084=-1108551,372643
EC00085=-1108551,372643
EC00086=-1108551,372643
EC00087=-1108551,372643
EC00088=-1108551,372643
EC00089=-1108551,372643
EC00090=-1108551,372643
EC00091=-1108551,372643
EC00092=-1108551,372643
EC00093=-1108551,372643
EC00094=-1108551,372643
EC00095=-1108551,372643
EC00096=-1108551,372643
EC00097=-1108551,372643
EC00098=-1108551,372643
EC00099=-1108551,372643
EC00100=-1108551,372643
EC00101=-1108551,372643
EC00102=-1108551,372643
EC00103=-1108551,372643
EC00104=-1108551,372643
EC00105=-1108551,372643
EC00106=-1108551,372643
EC00107=-1108551,372643
EC00108=-1108551,372643
EC00109=-1108550,372642
EC00110=-1108551,372643
EC00111=-1108551,372643
EC00112=-1108551,372643
EC00113=-1108551,372643
EC00114=-1108551,372643
EC00115=-1108551,372643
EC00116=-1108551,372643
EC00117=-1108551,372643
EC00118=-1108551,372643
EC00119=-1108551,372643
EC00120=-1108551,372643
EC00121=-1108551,372643
EC00122=-1108551,372643
EC00123=-1108551,372643
EC00124=-1108551,372642
EC00125=-1108551,372643
EC00126=-1108551,372643
EC00127=-1108551,372643
EC00128=-1108551,372643
EC00129=-1108551,372643
EC00130=-1108551,372643
EC00131=-1108551,372643
EC00132=-1108551,372643
EC00133=-1108551,372643
EC00134=-1108551,372643
EC00135=-1108551,372643
EC00136=-1108551,372643
EC00137=-1108551,372643
EC00138=-1108551,372643
EC00139=-1108551,372643
EC00140=-1108551,372643
EC00141=-1108551,372643
EC00142=-1108551,372643
EC00143=-1108551,372643
EC00144=-1108551,372643
EC00145=-1108551,372643
EC00146=-1108551,372643
EC00147=-1108551,372643
EC00148=-1108551,372643
EC00149=-1108551,372643
EC00150=-1108551,372643
EC00151=-1108551,372643
EC00152=-1108551,372643
EC00153=-1108551,372643
EC00154=-1108551,372643
EC00155=-1108551,372643
EC00156=-1108551,372643
EC00157=-1108551,372643
EC00158=-1108551,372643
EC00159=-1108551,372643
EC00160=-1108551,372643
EC00161=-1108551,372643
EC00162=-1108551,372643
EC00163=-1108551,372643
EC00164=-1108551,372643
EC00165=-1108551,372643
EC00166=-1108550,372643
EC00167=-1108550,372643
EC00168=-1108551,372643
EC00169=-1108551,372643
EC00170=-1108551,372643
EC00171=-1108551,372643
EC00172=-1108551,372643
EC00173=-1108551,372643
EC00174=-1108551,372643
EC00175=-1108551,372643
EC00176=-1108551,372643
EC00177=-1108551,372643
EC00178=-1108551,372643
EC00179=-1108551,372643
EC00180=-1108551,372643
EC00181=-1108551,372643
EC00182=-1108551,372643
EC00183=-1108551,372643
EC00184=-1108551,372643
EC00185=-1108551,372643
EC00186=-1108550,372643
EC00187=-1108551,372643
EC00188=-1108551,372643
EC00189=-1108551,372643
EC00190=-1108551,372643
EC00191=-1108551,372643
EC00192=-1108551,372643
EC00193=-1108551,372643
EC00194=-1108551,372643
EC00195=-1108551,372643
EC00196=-1108551,372643
EC00197=-1108551,372643
EC00198=-1108551,372643
EC00199=-1108551,372643
EC00200=-1108551,372643
EC00201=-1108551,372643
EC00202=1108549,-740306
EC00203=1108550,-740307
EC00204=1108551,-740307
EC00205=1108551,-740307
EC00206=1108551,-740307
EC00207=1108551,-740307
EC00208=1108551,-740307
EC00209=1108551,-740307
EC00210=1108551,-740307
EC00211=1108551,-740307
EC00212=1108551,-740307
EC00213=1108551,-740307
EC00214=1108551,-740307
EC00215=1108551,-740307
EC00216=1108551,-740307
EC00217=1108551,-740307
EC00218=1108551,-740307
EC00219=1108551,-740307
EC00220=1108551,-740307
EC00221=1108551,-740307
EC00222=1108551,-740307
EC00223=1108551,-740307
EC00224=1108551,-740307
EC00225=1108551,-740307
EC00226=1108551,-740307
EC00227=1108551,-740307
EC00228=1108551,-740307
EC00229=1108551,-740307
EC00230=1108551,-740307
EC00231=1108551,-740307
EC00232=1108551,-740307
EC00233=1108551,-740307
EC00234=1108551,-740307
EC00235=1108551,-740307
EC00236=1108551,-740307
EC00237=1108551,-740307
EC00238=1108551,-740307
EC00239=1108551,-740307
EC00240=1108551,-740307
EC00241=1108551,-740307
EC00242=1108551,-740307
EC00243=1108551,-740307
EC00244=1108551,-740307
EC00245=1108551,-740307
EC00246=1108551,-740307
EC00247=1108551,-740307
EC00248=1108551,-740307
EC00249=1108551,-740307
EC00250=1108551,-740307
EC00251=1108551,-740307
EC00252=1108551,-740307
EC00253=1108551,-740307
EC00254=1108551,-740307
EC00255=1108551,-740307
EC00256=1108551,-740307
EC00257=1108551,-740307
EC00258=1108551,-740307
EC00259=1108551,-740307
EC00260=1108551,-740307
EC00261=1108551,-740307
EC00262=1108550,-740307
EC00263=1108551,-740307
EC00264=1108551,-740307
EC00265=1108551,-740307
EC00266=1108551,-740307
EC00267=1108551,-740307
EC00268=1108551,-740307
EC00269=1108551,-740307
EC00270=1108551,-740307
EC00271=1108551,-740307
EC00272=1108551,-740307
EC00273=1108551,-740307
EC00274=1108551,-740307
EC00275=1108551,-740307
EC00276=1108551,-740307
EC00277=1108551,-740307
EC00278=1108551,-740307
EC00279=1108551,-740307
EC00280=1108551,-740307
EC00281=1108551,-740307
EC00282=1108551,-740307
EC00283=1108551,-740307
EC00284=1108551,-740307
EC00285=1108551,-740307
EC00286=1108551,-740307
EC00287=1108551,-740307
EC00288=1108551,-740307
EC00289=1108551,-740307
EC00290=1108551,-740307
EC00291=1108550,-740307
EC00292=1108550,-740307
EC00293=1108550,-740307
EC00294=1108550,-740307
EC00295=1108550,-740307
EC00296=1108551,-740307
EC00297=1108551,-740307
EC00298=1108551,-740307
EC00299=1108551,-740307
EC00300=1108551,-740307
EC00301=1108551,-740307
EC00302=1108551,-740307
EC00303=1108551,-740307
EC00304=1108551,-740307
EC00305=1108549,-740307
EC00306=1108550,-740307
EC00307=1108550,-740307
EC00308=1108550,-740307
EC00309=1108550,-740307
EC00310=1108550,-740307
EC00311=1108551,-740307
EC00312=1108549,-740308
EC00313=1108549,-740308
EC00314=1108549,-740308
EC00315=1108549,-740308
EC00316=1108549,-740308
EC00317=1108549,-740308
EC00318=1108551,-740307
EC00319=1108551,-740307
EC00320=1108551,-740307
EC00321=1108551,-740307
EC00322=1108551,-740307
EC00323=1108551,-740307
EC00324=1108551,-740307
EC00325=1108551,-740307
EC00326=1108551,-740307
EC00327=1108548,-740307
EC00328=1108550,-740308
EC00329=1108551,-740307
EC00330=1108551,-740307
EC00331=1108551,-740307
EC00332=1108551,-740307
EC00333=1108551,-740307
EC00334=1108551,-740307
EC00335=1108551,-740307
EC00336=1108551,-740307
EC00337=1108551,-740307
EC00338=1108551,-740307
EC00339=1108551,-740307
EC00340=1108551,-740307
EC00341=1108551,-740307
EC00342=1108551,-740307
EC00343=1108551,-740307
EC00344=1108551,-740307
EC00345=1108551,-740307
EC00346=1108551,-740307
EC00347=1108551,-740307
EC00348=1108551,-740307
EC00349=1108551,-740307
EC00350=1108551,-740307
EC00351=1108551,-740307
EC00352=1108551,-740307
EC00353=1108551,-740307
EC00354=1108551,-740307
EC00355=1108551,-740307
EC00356=1108551,-740307
EC00357=1108551,-740307
EC00358=1108551,-740307
EC00359=1108551,-740307
EC00360=1108551,-740307
EC00361=1108551,-740307
EC00362=1108551,-740307
EC00363=1108551,-740307
EC00364=1108551,-740307
EC00365=1108551,-740307
EC00366=1108551,-740307
EC00367=1108551,-740307
EC00368=1108551,-740307
EC00369=1108551,-740307
EC00370=1108551,-740307
EC00371=1108551,-740307
EC00372=1108551,-740307
EC00373=1108551,-740307
EC00374=1108551,-740307
EC00375=1108551,-740307
EC00376=1108551,-740307
EC00377=1108551,-740307
EC00378=1108551,-740307
EC00379=1108551,-740307
EC00380=1108551,-740307
EC00381=1108550,-740306
EC00382=1108550,-740306
EC00383=1108550,-740306
EC00384=1108550,-740306
EC00385=1108550,-740306
EC00386=1108550,-740306
EC00387=1108551,-740307
EC00388=1108551,-740307
EC00389=1108551,-740307
EC00390=1108551,-740307
EC00391=1108551,-740307
EC00392=1108551,-740307
EC00393=1108551,-740307
EC00394=1108551,-740307
EC00395=1108551,-740307
EC00396=1108551,-740307
EC00397=1108551,-740307
EC00398=1108551,-740307
EC00399=1108551,-740307
EC00400=1108551,-740307
EC00401=1108551,-740307
EC00402=1108551,-740307
EC00403=1108551,-740307
EC00404=1108551,-740307
EC00405=1108551,-740307
EC00406=1108551,-740307
EC00407=1108551,-740307
EC00408=1108551,-740307
EC00409=1108551,-740307
EC00410=1108551,-740307
EC00411=1108551,-740307
EC00412=1108551,-740307
EC00413=1108551,-740307
EC00414=1108551,-740307
EC00415=1108551,-740307
EC00416=1108551,-740307
EC00417=1108551,-740307
EC00418=1108551,-740307
EC00419=1108551,-740307
EC00420=1108551,-740307
EC00421=1108551,-740307
EC00422=1108551,-740307
EC00423=1108551,-740307
EC00424=1108551,-740307
EC00425=1108551,-740307
EC00426=1108551,-740307
EC00427=1108551,-740307
EC00428=1108551,-740307
EC00429=1108551,-740307
EC00430=1108551,-740307
EC00431=1108551,-740307
EC00432=1108551,-740307
EC00433=1108551,-740307
EC00434=1108551,-740307
EC00435=1108551,-740307
EC00436=1108551,-740307
EC00437=1108551,-740307
EC00438=1108551,-740307
EC00439=1108551,-740307
EC00440=1108551,-740307
EC00441=1108551,-740307
EC00442=1108551,-740307
EC00443=1108551,-740307
EC00444=1108551,-740307
EC00445=1108551,-740307
EC00446=1108550,-740307
EC00447=1108551,-740307
EC00448=1108551,-740307
EC00449=1108551,-740307
EC00450=1108551,-740307
EC00451=1108551,-740307
EC00452=1108551,-740307
EC00453=1108551,-740307
EC00454=1108551,-740307
EC00455=1108551,-740307
EC00456=1108551,-740307
EC00457=1108551,-740307
EC00458=1108551,-740307
EC00459=1108551,-740307
EC00460=1108551,-740307
EC00461=1108551,-740307
EC00462=1108551,-740307
EC00463=1108551,-740307
EC00464=1108551,-740307
EC00465=1108551,-740307
EC00466=1108551,-740307
EC00467=1108551,-740307
EC00468=1108551,-740307
EC00469=1108551,-740307
EC00470=1108551,-740307
EC00471=1108551,-740307
EC00472=1108551,-740307
EC00473=1108551,-740307
EC00474=1108551,-740307
EC00475=1108550,-740307
EC00476=1108550,-740307
EC00477=1108550,-740307
EC00478=1108550,-740307
EC00479=1108550,-740307
EC00480=1108551,-740307
EC00481=1108551,-740307
EC00482=1108551,-740307
EC00483=1108551,-740307
EC00484=1108551,-740307
EC00485=1108551,-740307
EC00486=1108551,-740307
EC00487=1108551,-740307
EC00488=1108551,-740307
EC00489=1108551,-740307
EC00490=1108551,-740307
EC00491=1108551,-740307
EC00492=1108551,-740307
EC00493=1108551,-740307
EC00494=1108551,-740307
EC00495=1108551,-740307
EC00496=1108551,-740307
EC00497=1108551,-740307
EC00498=1108549,-740308
EC00499=1108549,-740308
EC00500=1108549,-740308
EC00501=1108549,-740308
EC00502=1108549,-740308
EC00503=1108549,-740308
EC00504=1108551,-740307
EC00505=1108551,-740307
EC00506=1108551,-740307
EC00507=1108551,-740307
EC00508=1108551,-740307
EC00509=1108551,-740307
EC00510=1108551,-740307
EC00511=1108551,-740307
EC00512=1108551,-740307
EC00513=1108548,-740307
EC00514=1108550,-740308
EC00515=1108551,-740307
EC00516=1108551,-740307
EC00517=1108551,-740307
EC00518=1108551,-740307
EC00519=1108551,-740307
EC00520=1108551,-740307
EC00521=1108551,-740307
EC00522=1108551,-740307
EC00523=1108551,-740307
EC00524=1108551,-740307
EC00525=1108551,-740307
EC00526=1108551,-740307
EC00527=1108551,-740307
EC00528=1108551,-740307
EC00529=1108551,-740307
EC00530=1108551,-740307
EC00531=1108551,-740307
EC00532=1108551,-740307
EC00533=1108551,-740307
EC00534=1108551,-740307
EC00535=1108551,-740307
EC00536=1108551,-740307
EC00537=1108551,-740307
EC00538=1108551,-740307
EC00539=1108551,-740307
EC00540=1108551,-740307
EC00541=1108551,-740307
EC00542=1108551,-740307
EC00543=1108551,-740307
EC00544=1108551,-740307
EC00545=1108551,-740307
EC00546=1108551,-740307
EC00547=1108551,-740307
EC00548=1108551,-740307
EC00549=1108551,-740307
EC00550=1108551,-740307
EC00551=1108551,-740307
EC00552=1108551,-740307
EC00553=1108551,-740307
EC00554=1108551,-740307
EC00555=1108551,-740307
EC00556=1108551,-740307
EC00557=1108551,-740307
EC00558=1108551,-740307
EC00559=1108551,-740307
EC00560=1108551,-740307
EC00561=1108551,-740307
EC00562=1108551,-740307
EC00563=1108551,-740307
EC00564=1108551,-740307
EC00565=1108551,-740307
EC00566=1108551,-740307
EC00567=1108551,-740307
EC00568=1108551,-740307
EC00569=1108551,-740307
EC00570=1108551,-740307
EC00571=1108551,-740307
EC00572=1108551,-740307
///POSTYPE BASE
///RECTAN
///RCONF 0,0,0,0,1,0,0,0,0,0,0,0,0,0,0,0,0,0,0,0,0,0,0,0
P00006=2.006,1.622,-0.565,0.0000,0.0000,0.0000
P00021=0.073,2.058,-0.109,0.0000,0.0000,0.0000
P00022=2.006,1.622,-0.565,0.0000,0.0000,0.0000
///RCONF 0,0,0,0,0,0,0,0,0,0,0,0,0,0,0,0,0,0,0,0,0,0,0,0
P00023=-2.957,-4.083,2.762,0.0000,0.0000,0.0000
P00024=-1.466,-0.226,-0.419,0.0000,0.0000,0.0000
P00025=3.643,0.007,-2.585,0.0000,0.0000,0.0000
P00026=2.644,0.055,-2.583,0.0000,0.0000,0.0000
P00027=2.278,0.099,-4.210,0.0000,0.0000,0.0000
P00028=-1.778,-0.182,-2.050,0.0000,0.0000,0.0000
P00029=1.749,4.006,-0.261,0.0000,0.0000,0.0000
P00030=-0.014,-0.768,0.131,0.0000,0.0000,0.0000
P00031=-0.170,0.039,-0.647,0.0000,0.0000,0.0000
P00032=-0.423,0.157,3.222,0.0000,0.0000,0.0000
P00033=0.854,-1.099,3.047,0.0000,0.0000,0.0000
P00041=-0.109,0.014,0.966,0.0000,0.0000,0.0000
P00042=-0.220,0.371,-0.613,0.0000,0.0000,0.0000
P00043=-0.179,-5.890,-3.227,0.0000,0.0000,0.0000
P00044=-8.560,-7.557,-5.232,0.0000,0.0000,0.0000
P00045=-8.836,-6.632,-1.438,0.0000,0.0000,0.0000
P00046=-7.725,-0.107,-2.878,0.0000,0.0000,0.0000
///RCONF 0,1,0,0,0,0,0,0,0,0,0,0,0,0,0,0,0,0,0,0,0,0,0,0
P00047=0.052,4.745,-6.175,0.0000,0.0000,0.0000
///RCONF 0,0,0,0,0,0,0,0,0,0,0,0,0,0,0,0,0,0,0,0,0,0,0,0
P00048=-10.315,0.035,-3.101,0.0000,0.0000,0.0000
P00049=-9.638,1.690,-2.627,0.0000,0.0000,0.0000
P00050=-0.123,2.174,-1.314,0.0000,0.0000,0.0000
P00051=-5.945,4.696,-10.293,0.0000,0.0000,0.0000
P00052=-0.153,5.586,-7.982,0.0000,0.0000,0.0000
P00053=0.015,-0.644,-4.942,0.0000,0.0000,0.0000
//INST
///DATE 2024/12/10 13:33
///ATTR SC,RW
///GROUP1 RB1,BS1
///GROUP2 ST1
NOP
'X2_100(P)(125,-90)
COMM PAUSE
COMM MOVJ C00000 BC00000 VJ=20.00  +MOVJ EC00000 VJ=20.00
COMM MOVJ C00001 BC00001 VJ=20.00  +MOVJ EC00001 VJ=20.00
COMM PAUSE
COMM PAUSE
COMM '
COMM MOVJ C00002 BC00002 VJ=100.00  +MOVJ EC00002 VJ=100.00
COMM MOVJ C00003 BC00003 VJ=100.00  +MOVJ EC00003 VJ=100.00
COMM '
COMM MOVJ C00004 BC00004 VJ=100.00  +MOVJ EC00004 VJ=100.00
COMM MOVJ C00005 BC00005 VJ=100.00  +MOVJ EC00005 VJ=100.00
COMM MOVJ C00006 BC00006 VJ=100.00  +MOVJ EC00006 VJ=100.00
COMM MOVJ C00007 BC00007 VJ=100.00  +MOVJ EC00007 VJ=100.00
COMM MOVJ C00008 BC00008 VJ=100.00  +MOVJ EC00008 VJ=100.00
COMM 'Path S3336
COMM SFTOF3D
COMM MOVJ C00009 BC00009 VJ=100.00  +MOVJ EC00009 VJ=100.00
COMM MOVL C00010 BC00010 V=800.0  +MOVJ EC00010 VJ=100.00
COMM SMOVL C00011 BC00011 V=166.7  +MOVJ EC00011
COMM SREFP 3 C00012 BC00012  +REFP EC00012
COMM CALL JOB:SEARCH-R1-S13D
COMM SET P021 P006
COMM SFTON3D P021
COMM SMOVL C00013 BC00013 V=166.7  +MOVJ EC00013
COMM SREFP 3 C00014 BC00014  +REFP EC00014
COMM CALL JOB:SEARCH-R1-S13D
COMM SET P021 P006
COMM SFTON3D P021
COMM SMOVL C00015 BC00015 V=166.7  +MOVJ EC00015
COMM MOVL C00016 BC00016 V=1000.0  +MOVJ EC00016 VJ=100.00
COMM 'EndPath S3336
COMM 'Path S3337
COMM SFTOF3D
COMM MOVJ C00017 BC00017 VJ=100.00  +MOVJ EC00017 VJ=100.00
COMM MOVL C00018 BC00018 V=800.0  +MOVJ EC00018 VJ=100.00
COMM SMOVL C00019 BC00019 V=166.7  +MOVJ EC00019
COMM SREFP 3 C00020 BC00020  +REFP EC00020
COMM CALL JOB:SEARCH-R1-S13D
COMM SET P022 P006
COMM SFTON3D P022
COMM SMOVL C00021 BC00021 V=166.7  +MOVJ EC00021
COMM SREFP 3 C00022 BC00022  +REFP EC00022
COMM CALL JOB:SEARCH-R1-S13D
COMM SET P022 P006
COMM SFTON3D P022
COMM SMOVL C00023 BC00023 V=166.7  +MOVJ EC00023
COMM MOVL C00024 BC00024 V=1000.0  +MOVJ EC00024 VJ=100.00
COMM 'EndPath S3337
COMM 'Path S3338
COMM SFTOF3D
COMM MOVJ C00025 BC00025 VJ=100.00  +MOVJ EC00025 VJ=100.00
COMM MOVL C00026 BC00026 V=800.0  +MOVJ EC00026 VJ=100.00
COMM SMOVL C00027 BC00027 V=166.7  +MOVJ EC00027
COMM SREFP 3 C00028 BC00028  +REFP EC00028
COMM CALL JOB:SEARCH-R1-S13D
COMM SET P023 P006
COMM SFTON3D P023
COMM SMOVL C00029 BC00029 V=166.7  +MOVJ EC00029
COMM SREFP 3 C00030 BC00030  +REFP EC00030
COMM CALL JOB:SEARCH-R1-S13D
COMM SET P023 P006
COMM SFTON3D P023
COMM SMOVL C00031 BC00031 V=166.7  +MOVJ EC00031
COMM MOVL C00032 BC00032 V=1000.0  +MOVJ EC00032 VJ=100.00
COMM 'EndPath S3338
COMM MOVJ C00033 BC00033 VJ=100.00  +MOVJ EC00033 VJ=100.00
COMM 'Path S3339
COMM SFTOF3D
COMM MOVJ C00034 BC00034 VJ=100.00  +MOVJ EC00034 VJ=100.00
COMM MOVL C00035 BC00035 V=800.0  +MOVJ EC00035 VJ=100.00
COMM SMOVL C00036 BC00036 V=166.7  +MOVJ EC00036
COMM SREFP 3 C00037 BC00037  +REFP EC00037
COMM CALL JOB:SEARCH-R1-S13D
COMM SET P024 P006
COMM SFTON3D P024
COMM SMOVL C00038 BC00038 V=166.7  +MOVJ EC00038
COMM SREFP 3 C00039 BC00039  +REFP EC00039
COMM CALL JOB:SEARCH-R1-S13D
COMM SET P024 P006
COMM SFTON3D P024
COMM SMOVL C00040 BC00040 V=166.7  +MOVJ EC00040
COMM MOVL C00041 BC00041 V=1000.0  +MOVJ EC00041 VJ=100.00
COMM 'EndPath S3339
COMM 'Path S3341
COMM SFTOF3D
COMM MOVJ C00042 BC00042 VJ=100.00  +MOVJ EC00042 VJ=100.00
COMM MOVL C00043 BC00043 V=800.0  +MOVJ EC00043 VJ=100.00
COMM SMOVL C00044 BC00044 V=166.7  +MOVJ EC00044
COMM SREFP 3 C00045 BC00045  +REFP EC00045
COMM CALL JOB:SEARCH-R1-S13D
COMM SET P025 P006
COMM SFTON3D P025
COMM SMOVL C00046 BC00046 V=166.7  +MOVJ EC00046
COMM SREFP 3 C00047 BC00047  +REFP EC00047
COMM CALL JOB:SEARCH-R1-S13D
COMM SET P025 P006
COMM SFTON3D P025
COMM SMOVL C00048 BC00048 V=166.7  +MOVJ EC00048
COMM MOVL C00049 BC00049 V=1000.0  +MOVJ EC00049 VJ=100.00
COMM 'EndPath S3341
COMM 'Path S3343
COMM SFTOF3D
COMM MOVJ C00050 BC00050 VJ=100.00  +MOVJ EC00050 VJ=100.00
COMM MOVL C00051 BC00051 V=800.0  +MOVJ EC00051 VJ=100.00
COMM SMOVL C00052 BC00052 V=166.7  +MOVJ EC00052
COMM SREFP 3 C00053 BC00053  +REFP EC00053
COMM CALL JOB:SEARCH-R1-S13D
COMM SET P026 P006
COMM SFTON3D P026
COMM SMOVL C00054 BC00054 V=166.7  +MOVJ EC00054
COMM SREFP 3 C00055 BC00055  +REFP EC00055
COMM CALL JOB:SEARCH-R1-S13D
COMM SET P026 P006
COMM SFTON3D P026
COMM SMOVL C00056 BC00056 V=166.7  +MOVJ EC00056
COMM MOVL C00057 BC00057 V=1000.0  +MOVJ EC00057 VJ=100.00
COMM 'EndPath S3343
COMM MOVJ C00058 BC00058 VJ=100.00  +MOVJ EC00058 VJ=100.00
COMM 'Path S3345
COMM SFTOF3D
COMM MOVJ C00059 BC00059 VJ=100.00  +MOVJ EC00059 VJ=100.00
COMM MOVL C00060 BC00060 V=800.0  +MOVJ EC00060 VJ=100.00
COMM SMOVL C00061 BC00061 V=166.7  +MOVJ EC00061
COMM SREFP 3 C00062 BC00062  +REFP EC00062
COMM CALL JOB:SEARCH-R1-S13D
COMM SET P027 P006
COMM SFTON3D P027
COMM SMOVL C00063 BC00063 V=166.7  +MOVJ EC00063
COMM SREFP 3 C00064 BC00064  +REFP EC00064
COMM CALL JOB:SEARCH-R1-S13D
COMM SET P027 P006
COMM SFTON3D P027
COMM SMOVL C00065 BC00065 V=166.7  +MOVJ EC00065
COMM MOVL C00066 BC00066 V=1000.0  +MOVJ EC00066 VJ=100.00
COMM 'EndPath S3345
COMM MOVJ C00067 BC00067 VJ=100.00  +MOVJ EC00067 VJ=100.00
COMM 'Path S3347
COMM SFTOF3D
COMM MOVJ C00068 BC00068 VJ=100.00  +MOVJ EC00068 VJ=100.00
COMM MOVL C00069 BC00069 V=800.0  +MOVJ EC00069 VJ=100.00
COMM SMOVL C00070 BC00070 V=166.7  +MOVJ EC00070
COMM SREFP 3 C00071 BC00071  +REFP EC00071
COMM CALL JOB:SEARCH-R1-S13D
COMM SET P028 P006
COMM SFTON3D P028
COMM SMOVL C00072 BC00072 V=166.7  +MOVJ EC00072
COMM SREFP 3 C00073 BC00073  +REFP EC00073
COMM CALL JOB:SEARCH-R1-S13D
COMM SET P028 P006
COMM SFTON3D P028
COMM SMOVL C00074 BC00074 V=166.7  +MOVJ EC00074
COMM MOVL C00075 BC00075 V=1000.0  +MOVJ EC00075 VJ=100.00
COMM 'EndPath S3347
COMM 'Path S3349
COMM SFTOF3D
COMM MOVJ C00076 BC00076 VJ=100.00  +MOVJ EC00076 VJ=100.00
COMM MOVL C00077 BC00077 V=800.0  +MOVJ EC00077 VJ=100.00
COMM SMOVL C00078 BC00078 V=166.7  +MOVJ EC00078
COMM SREFP 3 C00079 BC00079  +REFP EC00079
COMM CALL JOB:SEARCH-R1-S13D
COMM SET P029 P006
COMM SFTON3D P029
COMM SMOVL C00080 BC00080 V=166.7  +MOVJ EC00080
COMM SREFP 3 C00081 BC00081  +REFP EC00081
COMM CALL JOB:SEARCH-R1-S13D
COMM SET P029 P006
COMM SFTON3D P029
COMM SMOVL C00082 BC00082 V=166.7  +MOVJ EC00082
COMM MOVL C00083 BC00083 V=1000.0  +MOVJ EC00083 VJ=100.00
COMM 'EndPath S3349
COMM 'Path S3350
COMM SFTOF3D
COMM MOVJ C00084 BC00084 VJ=100.00  +MOVJ EC00084 VJ=100.00
COMM MOVL C00085 BC00085 V=800.0  +MOVJ EC00085 VJ=100.00
COMM SMOVL C00086 BC00086 V=166.7  +MOVJ EC00086
COMM SREFP 3 C00087 BC00087  +REFP EC00087
COMM CALL JOB:SEARCH-R1-S13D
COMM SET P030 P006
COMM SFTON3D P030
COMM SMOVL C00088 BC00088 V=166.7  +MOVJ EC00088
COMM SREFP 3 C00089 BC00089  +REFP EC00089
COMM CALL JOB:SEARCH-R1-S13D
COMM SET P030 P006
COMM SFTON3D P030
COMM SMOVL C00090 BC00090 V=166.7  +MOVJ EC00090
COMM SMOVL C00091 BC00091 V=166.7  +MOVJ EC00091
COMM SREFP 3 C00092 BC00092  +REFP EC00092
COMM CALL JOB:SEARCH-R1-S13D
COMM SET P030 P006
COMM SFTON3D P030
COMM SMOVL C00093 BC00093 V=166.7  +MOVJ EC00093
COMM MOVL C00094 BC00094 V=1000.0  +MOVJ EC00094 VJ=100.00
COMM 'EndPath S3350
COMM 'Path S3351
COMM SFTOF3D
COMM MOVJ C00095 BC00095 VJ=100.00  +MOVJ EC00095 VJ=100.00
COMM MOVL C00096 BC00096 V=800.0  +MOVJ EC00096 VJ=100.00
COMM SMOVL C00097 BC00097 V=166.7  +MOVJ EC00097
COMM SREFP 3 C00098 BC00098  +REFP EC00098
COMM CALL JOB:SEARCH-R1-S13D
COMM SET P031 P006
COMM SFTON3D P031
COMM SMOVL C00099 BC00099 V=166.7  +MOVJ EC00099
COMM SREFP 3 C00100 BC00100  +REFP EC00100
COMM CALL JOB:SEARCH-R1-S13D
COMM SET P031 P006
COMM SFTON3D P031
COMM SMOVL C00101 BC00101 V=166.7  +MOVJ EC00101
COMM MOVL C00102 BC00102 V=1000.0  +MOVJ EC00102 VJ=100.00
COMM 'EndPath S3351
COMM MOVJ C00103 BC00103 VJ=100.00  +MOVJ EC00103 VJ=100.00
COMM 'Path S3352
COMM SFTOF3D
COMM MOVJ C00104 BC00104 VJ=100.00  +MOVJ EC00104 VJ=100.00
COMM MOVL C00105 BC00105 V=800.0  +MOVJ EC00105 VJ=100.00
COMM SMOVL C00106 BC00106 V=166.7  +MOVJ EC00106
COMM SREFP 3 C00107 BC00107  +REFP EC00107
COMM CALL JOB:SEARCH-R1-S13D
COMM SET P032 P006
COMM SFTON3D P032
COMM SMOVL C00108 BC00108 V=166.7  +MOVJ EC00108
COMM SREFP 3 C00109 BC00109  +REFP EC00109
COMM CALL JOB:SEARCH-R1-S13D
COMM SET P032 P006
COMM SFTON3D P032
COMM SMOVL C00110 BC00110 V=166.7  +MOVJ EC00110
COMM MOVL C00111 BC00111 V=1000.0  +MOVJ EC00111 VJ=100.00
COMM 'EndPath S3352
COMM 'Path S3353
COMM SFTOF3D
COMM MOVJ C00112 BC00112 VJ=100.00  +MOVJ EC00112 VJ=100.00
COMM MOVL C00113 BC00113 V=800.0  +MOVJ EC00113 VJ=100.00
COMM SMOVL C00114 BC00114 V=166.7  +MOVJ EC00114
COMM SREFP 3 C00115 BC00115  +REFP EC00115
COMM CALL JOB:SEARCH-R1-S13D
COMM SET P033 P006
COMM SFTON3D P033
COMM SMOVL C00116 BC00116 V=166.7  +MOVJ EC00116
COMM SREFP 3 C00117 BC00117  +REFP EC00117
COMM CALL JOB:SEARCH-R1-S13D
COMM SET P033 P006
COMM SFTON3D P033
COMM SMOVL C00118 BC00118 V=166.7  +MOVJ EC00118
COMM MOVL C00119 BC00119 V=1000.0  +MOVJ EC00119 VJ=100.00
COMM 'EndPath S3353
COMM MOVJ C00120 BC00120 VJ=100.00  +MOVJ EC00120 VJ=100.00
COMM MOVJ C00121 BC00121 VJ=100.00  +MOVJ EC00121 VJ=100.00
COMM 'Path W3292
COMM SFTOF3D
COMM SFTON3D P021
COMM MOVJ C00122 BC00122 VJ=100.00  +MOVJ EC00122 VJ=100.00
COMM SMOVL C00123 BC00123 V=800.0  +MOVJ EC00123
COMM SMOVL C00124 BC00124 V=166.7 PL=0  +MOVJ EC00124
COMM MACRO1 MJ#(0) ARGF9
COMM ARCON
COMM SMOVL C00125 BC00125 V=11.7  +MOVJ EC00125
COMM SMOVL C00126 BC00126 V=11.7  +MOVJ EC00126
COMM SMOVL C00127 BC00127 V=11.7  +MOVJ EC00127
COMM ARCOF
COMM SMOVL C00128 BC00128 V=800.0  +MOVJ EC00128
COMM SMOVL C00129 BC00129 V=1000.0  +MOVJ EC00129
COMM SFTOF3D
COMM 'EndPath W3292
COMM 'Path W3293
COMM SFTOF3D
COMM SFTON3D P022
COMM MOVJ C00130 BC00130 VJ=100.00  +MOVJ EC00130 VJ=100.00
COMM SMOVL C00131 BC00131 V=800.0  +MOVJ EC00131
COMM SMOVL C00132 BC00132 V=166.7 PL=0  +MOVJ EC00132
COMM ARCON
COMM SMOVL C00133 BC00133 V=11.7  +MOVJ EC00133
COMM ARCOF
COMM SMOVL C00134 BC00134 V=800.0  +MOVJ EC00134
COMM SMOVL C00135 BC00135 V=1000.0  +MOVJ EC00135
COMM SFTOF3D
COMM 'EndPath W3293
COMM 'Path W3294
COMM SFTOF3D
COMM SFTON3D P023
COMM MOVJ C00136 BC00136 VJ=100.00  +MOVJ EC00136 VJ=100.00
COMM SMOVL C00137 BC00137 V=800.0  +MOVJ EC00137
COMM SMOVL C00138 BC00138 V=166.7 PL=0  +MOVJ EC00138
COMM ARCON
COMM SMOVL C00139 BC00139 V=11.7  +MOVJ EC00139
COMM ARCOF
COMM SMOVL C00140 BC00140 V=800.0  +MOVJ EC00140
COMM SMOVL C00141 BC00141 V=1000.0  +MOVJ EC00141
COMM SFTOF3D
COMM 'EndPath W3294
COMM '
COMM MOVJ C00142 BC00142 VJ=100.00  +MOVJ EC00142 VJ=100.00
COMM 'Path W3340
COMM SFTOF3D
COMM SFTON3D P024
COMM MOVJ C00143 BC00143 VJ=100.00  +MOVJ EC00143 VJ=100.00
COMM SMOVL C00144 BC00144 V=800.0  +MOVJ EC00144
COMM SMOVL C00145 BC00145 V=150.0 PL=0  +MOVJ EC00145
COMM ARCON
COMM SMOVL C00146 BC00146 V=11.7  +MOVJ EC00146
COMM SMOVL C00147 BC00147 V=11.7  +MOVJ EC00147
COMM SMOVL C00148 BC00148 V=11.7  +MOVJ EC00148
COMM ARCOF
COMM SMOVL C00149 BC00149 V=800.0  +MOVJ EC00149
COMM SMOVL C00150 BC00150 V=1000.0  +MOVJ EC00150
COMM SFTOF3D
COMM 'EndPath W3340
COMM 'Path W3342
COMM SFTOF3D
COMM SFTON3D P025
COMM MOVJ C00151 BC00151 VJ=100.00  +MOVJ EC00151 VJ=100.00
COMM SMOVL C00152 BC00152 V=800.0  +MOVJ EC00152
COMM SMOVL C00153 BC00153 V=150.0 PL=0  +MOVJ EC00153
COMM ARCON
COMM SMOVL C00154 BC00154 V=11.7  +MOVJ EC00154
COMM ARCOF
COMM SMOVL C00155 BC00155 V=800.0  +MOVJ EC00155
COMM SMOVL C00156 BC00156 V=1000.0  +MOVJ EC00156
COMM SFTOF3D
COMM 'EndPath W3342
COMM 'Path W3344
COMM SFTOF3D
COMM SFTON3D P026
COMM MOVJ C00157 BC00157 VJ=100.00  +MOVJ EC00157 VJ=100.00
COMM SMOVL C00158 BC00158 V=800.0  +MOVJ EC00158
COMM SMOVL C00159 BC00159 V=150.0 PL=0  +MOVJ EC00159
COMM ARCON
COMM SMOVL C00160 BC00160 V=11.7  +MOVJ EC00160
COMM ARCOF
COMM SMOVL C00161 BC00161 V=800.0  +MOVJ EC00161
COMM SMOVL C00162 BC00162 V=1000.0  +MOVJ EC00162
COMM SFTOF3D
COMM 'EndPath W3344
COMM '
COMM MOVJ C00163 BC00163 VJ=100.00  +MOVJ EC00163 VJ=100.00
COMM 'Path W3346
COMM SFTOF3D
COMM SFTON3D P027
COMM MOVJ C00164 BC00164 VJ=100.00  +MOVJ EC00164 VJ=100.00
COMM SMOVL C00165 BC00165 V=800.0  +MOVJ EC00165
COMM SMOVL C00166 BC00166 V=150.0 PL=0  +MOVJ EC00166
COMM ARCON
COMM SMOVL C00167 BC00167 V=11.7  +MOVJ EC00167
COMM ARCOF
COMM SMOVL C00168 BC00168 V=800.0  +MOVJ EC00168
COMM SMOVL C00169 BC00169 V=1000.0  +MOVJ EC00169
COMM SFTOF3D
COMM 'EndPath W3346
COMM 'Path W3348
COMM SFTOF3D
COMM SFTON3D P028
COMM MOVJ C00170 BC00170 VJ=100.00  +MOVJ EC00170 VJ=100.00
COMM SMOVL C00171 BC00171 V=800.0  +MOVJ EC00171
COMM SMOVL C00172 BC00172 V=150.0 PL=0  +MOVJ EC00172
COMM ARCON
COMM SMOVL C00173 BC00173 V=11.7  +MOVJ EC00173
COMM ARCOF
COMM SMOVL C00174 BC00174 V=800.0  +MOVJ EC00174
COMM SMOVL C00175 BC00175 V=1000.0  +MOVJ EC00175
COMM SFTOF3D
COMM 'EndPath W3348
COMM 'Path W3350
COMM SFTOF3D
COMM SFTON3D P029
COMM MOVJ C00176 BC00176 VJ=100.00  +MOVJ EC00176 VJ=100.00
COMM SMOVL C00177 BC00177 V=800.0  +MOVJ EC00177
COMM SMOVL C00178 BC00178 V=150.0 PL=0  +MOVJ EC00178
COMM ARCON
COMM SMOVL C00179 BC00179 V=11.7  +MOVJ EC00179
COMM SMOVL C00180 BC00180 V=11.7  +MOVJ EC00180
COMM ARCOF
COMM SMOVL C00181 BC00181 V=800.0  +MOVJ EC00181
COMM SMOVL C00182 BC00182 V=1000.0  +MOVJ EC00182
COMM SFTOF3D
COMM 'EndPath W3350
COMM MOVJ C00183 BC00183 VJ=100.00  +MOVJ EC00183 VJ=100.00
COMM '
COMM 'Path W3316
COMM SFTOF3D
COMM SFTON3D P031
COMM MOVJ C00184 BC00184 VJ=100.00  +MOVJ EC00184 VJ=100.00
COMM SMOVL C00185 BC00185 V=800.0  +MOVJ EC00185
COMM SMOVL C00186 BC00186 V=150.0 PL=0  +MOVJ EC00186
COMM MACRO1 MJ#(0) ARGF21
COMM ARCON
COMM SMOVL C00187 BC00187 V=10.0  +MOVJ EC00187
COMM SFTON3D P030
COMM SMOVL C00188 BC00188 V=10.0  +MOVJ EC00188
COMM SMOVL C00189 BC00189 V=10.0  +MOVJ EC00189
COMM ARCOF
COMM SMOVL C00190 BC00190 V=800.0  +MOVJ EC00190
COMM SMOVL C00191 BC00191 V=1000.0  +MOVJ EC00191
COMM SFTOF3D
COMM 'EndPath W3316
COMM MOVJ C00192 BC00192 VJ=100.00  +MOVJ EC00192 VJ=100.00
COMM '
COMM 'Path W3319
COMM SFTOF3D
COMM SFTON3D P032
COMM MOVJ C00193 BC00193 VJ=100.00  +MOVJ EC00193 VJ=100.00
COMM SMOVL C00194 BC00194 V=800.0  +MOVJ EC00194
COMM SMOVL C00195 BC00195 V=150.0 PL=0  +MOVJ EC00195
COMM ARCON
COMM SFTON3D P033
COMM SMOVL C00196 BC00196 V=9.2  +MOVJ EC00196
COMM ARCOF
COMM SMOVL C00197 BC00197 V=800.0  +MOVJ EC00197
COMM SMOVL C00198 BC00198 V=1000.0  +MOVJ EC00198
COMM SFTOF3D
COMM 'EndPath W3319
COMM MOVJ C00199 BC00199 VJ=100.00  +MOVJ EC00199 VJ=100.00
COMM MOVJ C00200 BC00200 VJ=100.00  +MOVJ EC00200 VJ=100.00
COMM '
COMM MOVJ C00201 BC00201 VJ=100.00  +MOVJ EC00201 VJ=100.00
CALL JOB:CLEAN-R1_KM_NEW
MOVJ C00202 BC00202 VJ=15.00  +MOVJ EC00202 VJ=100.00
MOVJ C00203 BC00203 VJ=20.00  +MOVJ EC00203 VJ=20.00
'
'Path S3355
SFTOF3D
MOVJ C00204 BC00204 VJ=15.00  +MOVJ EC00204 VJ=100.00
MOVL C00205 BC00205 V=800.0  +MOVJ EC00205 VJ=100.00
MOVL C00206 BC00206 V=800.0  +MOVJ EC00206 VJ=100.00
SMOVL C00207 BC00207 V=166.7  +MOVJ EC00207
SREFP 3 C00208 BC00208  +REFP EC00208
CALL JOB:SEARCH-R1-S13D
SET P041 P006
SFTON3D P041
SMOVL C00209 BC00209 V=166.7  +MOVJ EC00209
SREFP 3 C00210 BC00210  +REFP EC00210
CALL JOB:SEARCH-R1-S13D
SET P041 P006
SFTON3D P041
SMOVL C00211 BC00211 V=166.7  +MOVJ EC00211
MOVL C00212 BC00212 V=250.0  +MOVJ EC00212 VJ=100.00
'EndPath S3355
'Path S3356
SFTOF3D
MOVJ C00213 BC00213 VJ=100.00  +MOVJ EC00213 VJ=100.00
MOVL C00214 BC00214 V=800.0  +MOVJ EC00214 VJ=100.00
SMOVL C00215 BC00215 V=166.7  +MOVJ EC00215
SREFP 3 C00216 BC00216  +REFP EC00216
CALL JOB:SEARCH-R1-S13D
SET P042 P006
SFTON3D P042
SMOVL C00217 BC00217 V=166.7  +MOVJ EC00217
SREFP 3 C00218 BC00218  +REFP EC00218
CALL JOB:SEARCH-R1-S13D
SET P042 P006
SFTON3D P042
SMOVL C00219 BC00219 V=166.7  +MOVJ EC00219
MOVL C00220 BC00220 V=1000.0  +MOVJ EC00220 VJ=100.00
'EndPath S3356
MOVJ C00221 BC00221 VJ=100.00  +MOVJ EC00221 VJ=100.00
MOVJ C00222 BC00222 VJ=100.00  +MOVJ EC00222 VJ=100.00
'Path S3357
SFTOF3D
MOVJ C00223 BC00223 VJ=100.00  +MOVJ EC00223 VJ=100.00
MOVL C00224 BC00224 V=333.3  +MOVJ EC00224 VJ=100.00
SMOVL C00225 BC00225 V=166.7  +MOVJ EC00225
SREFP 3 C00226 BC00226  +REFP EC00226
CALL JOB:SEARCH-R1-S13D
SET P043 P006
SFTON3D P043
SMOVL C00227 BC00227 V=166.7  +MOVJ EC00227
SREFP 3 C00228 BC00228  +REFP EC00228
CALL JOB:SEARCH-R1-S13D
SET P043 P006
SFTON3D P043
MOVL C00229 BC00229 V=800.0  +MOVJ EC00229 VJ=100.00
MOVL C00230 BC00230 V=500.0  +MOVJ EC00230 VJ=100.00
'EndPath S3357
MOVJ C00231 BC00231 VJ=20.00  +MOVJ EC00231 VJ=100.00
'Path S3358
SFTOF3D
MOVJ C00232 BC00232 VJ=100.00  +MOVJ EC00232 VJ=100.00
MOVL C00233 BC00233 V=800.0  +MOVJ EC00233 VJ=100.00
SMOVL C00234 BC00234 V=166.7  +MOVJ EC00234
SREFP 3 C00235 BC00235  +REFP EC00235
CALL JOB:SEARCH-R1-S13D
SET P044 P006
SFTON3D P044
SMOVL C00236 BC00236 V=166.7  +MOVJ EC00236
SREFP 3 C00237 BC00237  +REFP EC00237
CALL JOB:SEARCH-R1-S13D
SET P044 P006
SFTON3D P044
SMOVL C00238 BC00238 V=166.7  +MOVJ EC00238
MOVL C00239 BC00239 V=1000.0  +MOVJ EC00239 VJ=100.00
'EndPath S3358
'Path S3359
SFTOF3D
MOVJ C00240 BC00240 VJ=100.00  +MOVJ EC00240 VJ=100.00
MOVL C00241 BC00241 V=800.0  +MOVJ EC00241 VJ=100.00
SMOVL C00242 BC00242 V=166.7  +MOVJ EC00242
SREFP 3 C00243 BC00243  +REFP EC00243
CALL JOB:SEARCH-R1-S13D
SET P045 P006
SFTON3D P045
SMOVL C00244 BC00244 V=166.7  +MOVJ EC00244
SREFP 3 C00245 BC00245  +REFP EC00245
CALL JOB:SEARCH-R1-S13D
SET P045 P006
SFTON3D P045
SMOVL C00246 BC00246 V=166.7  +MOVJ EC00246
MOVL C00247 BC00247 V=1000.0  +MOVJ EC00247 VJ=100.00
'EndPath S3359
'Path S3360
SFTOF3D
MOVJ C00248 BC00248 VJ=100.00  +MOVJ EC00248 VJ=100.00
MOVL C00249 BC00249 V=800.0  +MOVJ EC00249 VJ=100.00
SMOVL C00250 BC00250 V=166.7  +MOVJ EC00250
SREFP 3 C00251 BC00251  +REFP EC00251
CALL JOB:SEARCH-R1-S13D
SET P046 P006
SFTON3D P046
SMOVL C00252 BC00252 V=166.7  +MOVJ EC00252
SREFP 3 C00253 BC00253  +REFP EC00253
CALL JOB:SEARCH-R1-S13D
SET P046 P006
SFTON3D P046
SMOVL C00254 BC00254 V=166.7  +MOVJ EC00254
MOVL C00255 BC00255 V=1000.0  +MOVJ EC00255 VJ=100.00
'EndPath S3360
MOVJ C00256 BC00256 VJ=100.00  +MOVJ EC00256 VJ=100.00
'Path S3361
SFTOF3D
MOVJ C00257 BC00257 VJ=25.00  +MOVJ EC00257 VJ=100.00
MOVL C00258 BC00258 V=800.0  +MOVJ EC00258 VJ=100.00
SMOVL C00259 BC00259 V=166.7  +MOVJ EC00259
SREFP 3 C00260 BC00260  +REFP EC00260
CALL JOB:SEARCH-R1-S13D
SET P047 P006
SFTON3D P047
SMOVL C00261 BC00261 V=166.7  +MOVJ EC00261
SREFP 3 C00262 BC00262  +REFP EC00262
CALL JOB:SEARCH-R1-S13D
SET P047 P006
SFTON3D P047
SMOVL C00263 BC00263 V=166.7  +MOVJ EC00263
MOVL C00264 BC00264 V=1000.0  +MOVJ EC00264 VJ=100.00
'EndPath S3361
'Path S3362
SFTOF3D
MOVJ C00265 BC00265 VJ=100.00  +MOVJ EC00265 VJ=100.00
MOVL C00266 BC00266 V=800.0  +MOVJ EC00266 VJ=100.00
SMOVL C00267 BC00267 V=166.7  +MOVJ EC00267
SREFP 3 C00268 BC00268  +REFP EC00268
CALL JOB:SEARCH-R1-S13D
SET P048 P006
SFTON3D P048
SMOVL C00269 BC00269 V=166.7  +MOVJ EC00269
SREFP 3 C00270 BC00270  +REFP EC00270
CALL JOB:SEARCH-R1-S13D
SET P048 P006
SFTON3D P048
SMOVL C00271 BC00271 V=166.7  +MOVJ EC00271
MOVL C00272 BC00272 V=1000.0  +MOVJ EC00272 VJ=100.00
'EndPath S3362
'Path S3363
SFTOF3D
MOVJ C00273 BC00273 VJ=100.00  +MOVJ EC00273 VJ=100.00
MOVL C00274 BC00274 V=800.0  +MOVJ EC00274 VJ=100.00
SMOVL C00275 BC00275 V=166.7  +MOVJ EC00275
SREFP 3 C00276 BC00276  +REFP EC00276
CALL JOB:SEARCH-R1-S13D
SET P049 P006
SFTON3D P049
SMOVL C00277 BC00277 V=166.7  +MOVJ EC00277
SREFP 3 C00278 BC00278  +REFP EC00278
CALL JOB:SEARCH-R1-S13D
SET P049 P006
SFTON3D P049
SMOVL C00279 BC00279 V=166.7  +MOVJ EC00279
MOVL C00280 BC00280 V=1000.0  +MOVJ EC00280 VJ=100.00
'EndPath S3363
'Path S3364
SFTOF3D
MOVJ C00281 BC00281 VJ=100.00  +MOVJ EC00281 VJ=100.00
MOVJ C00282 BC00282 VJ=25.00  +MOVJ EC00282 VJ=100.00
MOVL C00283 BC00283 V=800.0  +MOVJ EC00283 VJ=100.00
SMOVL C00284 BC00284 V=166.7  +MOVJ EC00284
SREFP 3 C00285 BC00285  +REFP EC00285
CALL JOB:SEARCH-R1-S13D
SET P050 P006
SFTON3D P050
SMOVL C00286 BC00286 V=166.7  +MOVJ EC00286
SREFP 3 C00287 BC00287  +REFP EC00287
CALL JOB:SEARCH-R1-S13D
SET P050 P006
SFTON3D P050
SMOVL C00288 BC00288 V=166.7  +MOVJ EC00288
'EndPath S3364
'Path S3365
SFTOF3D
MOVJ C00289 BC00289 VJ=100.00  +MOVJ EC00289 VJ=100.00
MOVL C00290 BC00290 V=800.0  +MOVJ EC00290 VJ=100.00
SMOVL C00291 BC00291 V=166.7  +MOVJ EC00291
SREFP 3 C00292 BC00292  +REFP EC00292
CALL JOB:SEARCH-R1-S13D
SET P051 P006
SFTON3D P051
SMOVL C00293 BC00293 V=166.7  +MOVJ EC00293
SREFP 3 C00294 BC00294  +REFP EC00294
CALL JOB:SEARCH-R1-S13D
SET P051 P006
SFTON3D P051
SMOVL C00295 BC00295 V=166.7  +MOVJ EC00295
MOVL C00296 BC00296 V=333.3  +MOVJ EC00296 VJ=100.00
'EndPath S3365
MOVJ C00297 BC00297 VJ=20.00  +MOVJ EC00297 VJ=100.00
'Path S3366
SFTOF3D
MOVJ C00298 BC00298 VJ=20.00  +MOVJ EC00298 VJ=100.00
MOVL C00299 BC00299 V=800.0  +MOVJ EC00299 VJ=100.00
SMOVL C00300 BC00300 V=166.7  +MOVJ EC00300
SREFP 3 C00301 BC00301  +REFP EC00301
CALL JOB:SEARCH-R1-S13D
SET P052 P006
SFTON3D P052
SMOVL C00302 BC00302 V=166.7  +MOVJ EC00302
SREFP 3 C00303 BC00303  +REFP EC00303
CALL JOB:SEARCH-R1-S13D
SET P052 P006
SFTON3D P052
SMOVL C00304 BC00304 V=166.7  +MOVJ EC00304
'EndPath S3366
'Path S3367
SFTOF3D
MOVL C00305 BC00305 V=800.0  +MOVJ EC00305 VJ=100.00
SMOVL C00306 BC00306 V=166.7  +MOVJ EC00306
SREFP 3 C00307 BC00307  +REFP EC00307
CALL JOB:SEARCH-R1-S13D
SET P053 P006
SFTON3D P053
SMOVL C00308 BC00308 V=166.7  +MOVJ EC00308
SREFP 3 C00309 BC00309  +REFP EC00309
CALL JOB:SEARCH-R1-S13D
SET P053 P006
SFTON3D P053
SMOVL C00310 BC00310 V=166.7  +MOVJ EC00310
SFTOF3D
MOVL C00311 BC00311 V=333.3  +MOVJ EC00311 VJ=100.00
'EndPath S3367
'
'Path W3331
SFTOF3D
SFTON3D P052
MOVJ C00312 BC00312 VJ=100.00  +MOVJ EC00312 VJ=100.00
SMOVL C00313 BC00313 V=800.0  +MOVJ EC00313
SMOVL C00314 BC00314 V=150.0 PL=0  +MOVJ EC00314
ARCON
SFTON3D P053
SMOVL C00315 BC00315 V=9.2  +MOVJ EC00315
ARCOF
SMOVL C00316 BC00316 V=800.0  +MOVJ EC00316
SMOVL C00317 BC00317 V=1000.0  +MOVJ EC00317
SFTOF3D
'EndPath W3331
MOVJ C00318 BC00318 VJ=100.00  +MOVJ EC00318 VJ=100.00
'
'Path W3335
SFTOF3D
SFTON3D P051
MOVJ C00319 BC00319 VJ=100.00  +MOVJ EC00319 VJ=100.00
SMOVL C00320 BC00320 V=800.0  +MOVJ EC00320
SMOVL C00321 BC00321 V=150.0 PL=0  +MOVJ EC00321
ARCON
SFTON3D P050
SMOVL C00322 BC00322 V=9.2  +MOVJ EC00322
ARCOF
SMOVL C00323 BC00323 V=416.7  +MOVJ EC00323
SMOVL C00324 BC00324 V=500.0  +MOVJ EC00324
SFTOF3D
'EndPath W3335
'
'Path W3326
SFTOF3D
SFTON3D P047
MOVJ C00325 BC00325 VJ=100.00  +MOVJ EC00325 VJ=100.00
SMOVL C00326 BC00326 V=800.0  +MOVJ EC00326
SMOVL C00327 BC00327 V=150.0 PL=0  +MOVJ EC00327
MACRO1 MJ#(0) ARGF9
ARCON
SMOVL C00328 BC00328 V=11.7  +MOVJ EC00328
ARCOF
SMOVL C00329 BC00329 V=800.0  +MOVJ EC00329
SMOVL C00330 BC00330 V=500.0  +MOVJ EC00330
SFTOF3D
'EndPath W3326
'Path W3327
SFTOF3D
SFTON3D P048
MOVJ C00331 BC00331 VJ=100.00  +MOVJ EC00331 VJ=100.00
SMOVL C00332 BC00332 V=800.0  +MOVJ EC00332
SMOVL C00333 BC00333 V=150.0 PL=0  +MOVJ EC00333
ARCON
SMOVL C00334 BC00334 V=11.7  +MOVJ EC00334
ARCOF
SMOVL C00335 BC00335 V=800.0  +MOVJ EC00335
SMOVL C00336 BC00336 V=1000.0  +MOVJ EC00336
SFTOF3D
'EndPath W3327
'Path W3328
SFTOF3D
SFTON3D P049
MOVJ C00337 BC00337 VJ=100.00  +MOVJ EC00337 VJ=100.00
SMOVL C00338 BC00338 V=800.0  +MOVJ EC00338
SMOVL C00339 BC00339 V=150.0 PL=0  +MOVJ EC00339
ARCON
SMOVL C00340 BC00340 V=11.7  +MOVJ EC00340
SMOVL C00341 BC00341 V=11.7  +MOVJ EC00341
ARCOF
SMOVL C00342 BC00342 V=333.3  +MOVJ EC00342
SMOVL C00343 BC00343 V=500.0  +MOVJ EC00343
SFTOF3D
'EndPath W3328
MOVJ C00344 BC00344 VJ=100.00  +MOVJ EC00344 VJ=100.00
'
'Path W3323
SFTOF3D
SFTON3D P044
MOVJ C00345 BC00345 VJ=20.00  +MOVJ EC00345 VJ=100.00
SMOVL C00346 BC00346 V=800.0  +MOVJ EC00346
SMOVL C00347 BC00347 V=150.0 PL=0  +MOVJ EC00347
ARCON
SMOVL C00348 BC00348 V=11.7  +MOVJ EC00348
SMOVL C00349 BC00349 V=11.7  +MOVJ EC00349
ARCOF
SMOVL C00350 BC00350 V=333.3  +MOVJ EC00350
SFTOF3D
'EndPath W3323
'Path W3324
SFTOF3D
SFTON3D P045
MOVJ C00351 BC00351 VJ=100.00  +MOVJ EC00351 VJ=100.00
SMOVL C00352 BC00352 V=800.0  +MOVJ EC00352
SMOVL C00353 BC00353 V=150.0 PL=0  +MOVJ EC00353
ARCON
SMOVL C00354 BC00354 V=11.7  +MOVJ EC00354
ARCOF
SMOVL C00355 BC00355 V=800.0  +MOVJ EC00355
SFTOF3D
'EndPath W3324
'Path W3325
SFTOF3D
SFTON3D P046
MOVJ C00356 BC00356 VJ=20.00  +MOVJ EC00356 VJ=100.00
SMOVL C00357 BC00357 V=800.0  +MOVJ EC00357
SMOVL C00358 BC00358 V=150.0 PL=0  +MOVJ EC00358
ARCON
SMOVL C00359 BC00359 V=11.7  +MOVJ EC00359
ARCOF
SMOVL C00360 BC00360 V=500.0  +MOVJ EC00360
SFTOF3D
'EndPath W3325
'
'
'Path W3320
SFTOF3D
SFTON3D P041
MOVJ C00361 BC00361 VJ=100.00  +MOVJ EC00361 VJ=100.00
SMOVL C00362 BC00362 V=800.0  +MOVJ EC00362
SMOVL C00363 BC00363 V=166.7 PL=0  +MOVJ EC00363
ARCON
SMOVL C00364 BC00364 V=11.7  +MOVJ EC00364
ARCOF
SMOVL C00365 BC00365 V=333.3  +MOVJ EC00365
SMOVL C00366 BC00366 V=500.0  +MOVJ EC00366
SFTOF3D
'EndPath W3320
'Path W3321
SFTOF3D
SFTON3D P042
MOVJ C00367 BC00367 VJ=100.00  +MOVJ EC00367 VJ=100.00
SMOVL C00368 BC00368 V=800.0  +MOVJ EC00368
SMOVL C00369 BC00369 V=166.7 PL=0  +MOVJ EC00369
ARCON
SMOVL C00370 BC00370 V=11.7  +MOVJ EC00370
ARCOF
SMOVL C00371 BC00371 V=800.0  +MOVJ EC00371
SFTOF3D
'EndPath W3321
'Path W3322
SFTOF3D
SFTON3D P043
MOVJ C00372 BC00372 VJ=100.00  +MOVJ EC00372 VJ=100.00
SMOVL C00373 BC00373 V=800.0  +MOVJ EC00373
SMOVL C00374 BC00374 V=166.7 PL=0  +MOVJ EC00374
ARCON
SMOVL C00375 BC00375 V=11.7  +MOVJ EC00375
SMOVL C00376 BC00376 V=11.7  +MOVJ EC00376
ARCOF
SMOVL C00377 BC00377 V=333.3  +MOVJ EC00377
SMOVL C00378 BC00378 V=500.0  +MOVJ EC00378
SFTOF3D
'EndPath W3322
MOVJ C00379 BC00379 VJ=20.00  +MOVJ EC00379 VJ=100.00
MOVJ C00380 BC00380 VJ=20.00  +MOVJ EC00380 VJ=100.00
PAUSE
MOVJ C00381 BC00381 VJ=20.00  +MOVJ EC00381 VJ=100.00
MOVJ C00382 BC00382 VJ=20.00  +MOVJ EC00382 VJ=100.00
MOVJ C00383 BC00383 VJ=20.00  +MOVJ EC00383 VJ=100.00
MOVJ C00384 BC00384 VJ=20.00  +MOVJ EC00384 VJ=20.00
MOVJ C00385 BC00385 VJ=20.00  +MOVJ EC00385 VJ=100.00
MOVJ C00386 BC00386 VJ=20.00  +MOVJ EC00386 VJ=20.00
CALL JOB:CLEAN-R1_KM_NEW
MOVJ C00387 BC00387 VJ=100.00  +MOVJ EC00387 VJ=100.00
'
'Path S3355
SFTOF3D
MOVJ C00388 BC00388 VJ=100.00  +MOVJ EC00388 VJ=100.00
MOVL C00389 BC00389 V=800.0  +MOVJ EC00389 VJ=100.00
MOVL C00390 BC00390 V=800.0  +MOVJ EC00390 VJ=100.00
SMOVL C00391 BC00391 V=166.7  +MOVJ EC00391
SREFP 3 C00392 BC00392  +REFP EC00392
CALL JOB:SEARCH-R1-S13D
SET P041 P006
SFTON3D P041
SMOVL C00393 BC00393 V=166.7  +MOVJ EC00393
SREFP 3 C00394 BC00394  +REFP EC00394
CALL JOB:SEARCH-R1-S13D
SET P041 P006
SFTON3D P041
SMOVL C00395 BC00395 V=166.7  +MOVJ EC00395
MOVL C00396 BC00396 V=1000.0  +MOVJ EC00396 VJ=100.00
'EndPath S3355
'Path S3356
SFTOF3D
MOVJ C00397 BC00397 VJ=100.00  +MOVJ EC00397 VJ=100.00
MOVL C00398 BC00398 V=800.0  +MOVJ EC00398 VJ=100.00
SMOVL C00399 BC00399 V=166.7  +MOVJ EC00399
SREFP 3 C00400 BC00400  +REFP EC00400
CALL JOB:SEARCH-R1-S13D
SET P042 P006
SFTON3D P042
SMOVL C00401 BC00401 V=166.7  +MOVJ EC00401
SREFP 3 C00402 BC00402  +REFP EC00402
CALL JOB:SEARCH-R1-S13D
SET P042 P006
SFTON3D P042
SMOVL C00403 BC00403 V=166.7  +MOVJ EC00403
MOVL C00404 BC00404 V=1000.0  +MOVJ EC00404 VJ=100.00
'EndPath S3356
MOVJ C00405 BC00405 VJ=100.00  +MOVJ EC00405 VJ=100.00
MOVJ C00406 BC00406 VJ=100.00  +MOVJ EC00406 VJ=100.00
'Path S3357
SFTOF3D
MOVJ C00407 BC00407 VJ=100.00  +MOVJ EC00407 VJ=100.00
MOVL C00408 BC00408 V=800.0  +MOVJ EC00408 VJ=100.00
SMOVL C00409 BC00409 V=166.7  +MOVJ EC00409
SREFP 3 C00410 BC00410  +REFP EC00410
CALL JOB:SEARCH-R1-S13D
SET P043 P006
SFTON3D P043
SMOVL C00411 BC00411 V=166.7  +MOVJ EC00411
SREFP 3 C00412 BC00412  +REFP EC00412
CALL JOB:SEARCH-R1-S13D
SET P043 P006
SFTON3D P043
MOVL C00413 BC00413 V=800.0  +MOVJ EC00413 VJ=100.00
MOVL C00414 BC00414 V=500.0  +MOVJ EC00414 VJ=100.00
'EndPath S3357
MOVJ C00415 BC00415 VJ=100.00  +MOVJ EC00415 VJ=100.00
'Path S3358
SFTOF3D
MOVJ C00416 BC00416 VJ=100.00  +MOVJ EC00416 VJ=100.00
MOVL C00417 BC00417 V=800.0  +MOVJ EC00417 VJ=100.00
SMOVL C00418 BC00418 V=166.7  +MOVJ EC00418
SREFP 3 C00419 BC00419  +REFP EC00419
CALL JOB:SEARCH-R1-S13D
SET P044 P006
SFTON3D P044
SMOVL C00420 BC00420 V=166.7  +MOVJ EC00420
SREFP 3 C00421 BC00421  +REFP EC00421
CALL JOB:SEARCH-R1-S13D
SET P044 P006
SFTON3D P044
SMOVL C00422 BC00422 V=166.7  +MOVJ EC00422
MOVL C00423 BC00423 V=1000.0  +MOVJ EC00423 VJ=100.00
'EndPath S3358
'Path S3359
SFTOF3D
MOVJ C00424 BC00424 VJ=100.00  +MOVJ EC00424 VJ=100.00
MOVL C00425 BC00425 V=800.0  +MOVJ EC00425 VJ=100.00
SMOVL C00426 BC00426 V=166.7  +MOVJ EC00426
SREFP 3 C00427 BC00427  +REFP EC00427
CALL JOB:SEARCH-R1-S13D
SET P045 P006
SFTON3D P045
SMOVL C00428 BC00428 V=166.7  +MOVJ EC00428
SREFP 3 C00429 BC00429  +REFP EC00429
CALL JOB:SEARCH-R1-S13D
SET P045 P006
SFTON3D P045
SMOVL C00430 BC00430 V=166.7  +MOVJ EC00430
MOVL C00431 BC00431 V=1000.0  +MOVJ EC00431 VJ=100.00
'EndPath S3359
'Path S3360
SFTOF3D
MOVJ C00432 BC00432 VJ=100.00  +MOVJ EC00432 VJ=100.00
MOVL C00433 BC00433 V=800.0  +MOVJ EC00433 VJ=100.00
SMOVL C00434 BC00434 V=166.7  +MOVJ EC00434
SREFP 3 C00435 BC00435  +REFP EC00435
CALL JOB:SEARCH-R1-S13D
SET P046 P006
SFTON3D P046
SMOVL C00436 BC00436 V=166.7  +MOVJ EC00436
SREFP 3 C00437 BC00437  +REFP EC00437
CALL JOB:SEARCH-R1-S13D
SET P046 P006
SFTON3D P046
SMOVL C00438 BC00438 V=166.7  +MOVJ EC00438
MOVL C00439 BC00439 V=1000.0  +MOVJ EC00439 VJ=100.00
'EndPath S3360
MOVJ C00440 BC00440 VJ=100.00  +MOVJ EC00440 VJ=100.00
'Path S3361
SFTOF3D
MOVJ C00441 BC00441 VJ=100.00  +MOVJ EC00441 VJ=100.00
MOVL C00442 BC00442 V=800.0  +MOVJ EC00442 VJ=100.00
SMOVL C00443 BC00443 V=166.7  +MOVJ EC00443
SREFP 3 C00444 BC00444  +REFP EC00444
CALL JOB:SEARCH-R1-S13D
SET P047 P006
SFTON3D P047
SMOVL C00445 BC00445 V=166.7  +MOVJ EC00445
SREFP 3 C00446 BC00446  +REFP EC00446
CALL JOB:SEARCH-R1-S13D
SET P047 P006
SFTON3D P047
SMOVL C00447 BC00447 V=166.7  +MOVJ EC00447
MOVL C00448 BC00448 V=1000.0  +MOVJ EC00448 VJ=100.00
'EndPath S3361
'Path S3362
SFTOF3D
MOVJ C00449 BC00449 VJ=100.00  +MOVJ EC00449 VJ=100.00
MOVL C00450 BC00450 V=800.0  +MOVJ EC00450 VJ=100.00
SMOVL C00451 BC00451 V=166.7  +MOVJ EC00451
SREFP 3 C00452 BC00452  +REFP EC00452
CALL JOB:SEARCH-R1-S13D
SET P048 P006
SFTON3D P048
SMOVL C00453 BC00453 V=166.7  +MOVJ EC00453
SREFP 3 C00454 BC00454  +REFP EC00454
CALL JOB:SEARCH-R1-S13D
SET P048 P006
SFTON3D P048
SMOVL C00455 BC00455 V=166.7  +MOVJ EC00455
MOVL C00456 BC00456 V=1000.0  +MOVJ EC00456 VJ=100.00
'EndPath S3362
'Path S3363
SFTOF3D
MOVJ C00457 BC00457 VJ=100.00  +MOVJ EC00457 VJ=100.00
MOVL C00458 BC00458 V=800.0  +MOVJ EC00458 VJ=100.00
SMOVL C00459 BC00459 V=166.7  +MOVJ EC00459
SREFP 3 C00460 BC00460  +REFP EC00460
CALL JOB:SEARCH-R1-S13D
SET P049 P006
SFTON3D P049
SMOVL C00461 BC00461 V=166.7  +MOVJ EC00461
SREFP 3 C00462 BC00462  +REFP EC00462
CALL JOB:SEARCH-R1-S13D
SET P049 P006
SFTON3D P049
SMOVL C00463 BC00463 V=166.7  +MOVJ EC00463
MOVL C00464 BC00464 V=1000.0  +MOVJ EC00464 VJ=100.00
'EndPath S3363
'Path S3364
SFTOF3D
MOVJ C00465 BC00465 VJ=100.00  +MOVJ EC00465 VJ=100.00
MOVJ C00466 BC00466 VJ=100.00  +MOVJ EC00466 VJ=100.00
MOVL C00467 BC00467 V=800.0  +MOVJ EC00467 VJ=100.00
SMOVL C00468 BC00468 V=166.7  +MOVJ EC00468
SREFP 3 C00469 BC00469  +REFP EC00469
CALL JOB:SEARCH-R1-S13D
SET P050 P006
SFTON3D P050
SMOVL C00470 BC00470 V=166.7  +MOVJ EC00470
SREFP 3 C00471 BC00471  +REFP EC00471
CALL JOB:SEARCH-R1-S13D
SET P050 P006
SFTON3D P050
SMOVL C00472 BC00472 V=166.7  +MOVJ EC00472
'EndPath S3364
'Path S3365
SFTOF3D
MOVJ C00473 BC00473 VJ=100.00  +MOVJ EC00473 VJ=100.00
MOVL C00474 BC00474 V=800.0  +MOVJ EC00474 VJ=100.00
SMOVL C00475 BC00475 V=166.7  +MOVJ EC00475
SREFP 3 C00476 BC00476  +REFP EC00476
CALL JOB:SEARCH-R1-S13D
SET P051 P006
SFTON3D P051
SMOVL C00477 BC00477 V=166.7  +MOVJ EC00477
SREFP 3 C00478 BC00478  +REFP EC00478
CALL JOB:SEARCH-R1-S13D
SET P051 P006
SFTON3D P051
SMOVL C00479 BC00479 V=166.7  +MOVJ EC00479
MOVL C00480 BC00480 V=1000.0  +MOVJ EC00480 VJ=100.00
'EndPath S3365
MOVJ C00481 BC00481 VJ=100.00  +MOVJ EC00481 VJ=100.00
'Path S3366
SFTOF3D
MOVJ C00482 BC00482 VJ=100.00  +MOVJ EC00482 VJ=100.00
MOVL C00483 BC00483 V=800.0  +MOVJ EC00483 VJ=100.00
SMOVL C00484 BC00484 V=166.7  +MOVJ EC00484
SREFP 3 C00485 BC00485  +REFP EC00485
CALL JOB:SEARCH-R1-S13D
SET P052 P006
SFTON3D P052
SMOVL C00486 BC00486 V=166.7  +MOVJ EC00486
SREFP 3 C00487 BC00487  +REFP EC00487
CALL JOB:SEARCH-R1-S13D
SET P052 P006
SFTON3D P052
SMOVL C00488 BC00488 V=166.7  +MOVJ EC00488
MOVL C00489 BC00489 V=1000.0  +MOVJ EC00489 VJ=100.00
'EndPath S3366
'Path S3367
SFTOF3D
MOVJ C00490 BC00490 VJ=100.00  +MOVJ EC00490 VJ=100.00
MOVL C00491 BC00491 V=800.0  +MOVJ EC00491 VJ=100.00
SMOVL C00492 BC00492 V=166.7  +MOVJ EC00492
SREFP 3 C00493 BC00493  +REFP EC00493
CALL JOB:SEARCH-R1-S13D
SET P053 P006
SFTON3D P053
SMOVL C00494 BC00494 V=166.7  +MOVJ EC00494
SREFP 3 C00495 BC00495  +REFP EC00495
CALL JOB:SEARCH-R1-S13D
SET P053 P006
SFTON3D P053
SMOVL C00496 BC00496 V=166.7  +MOVJ EC00496
SFTOF3D
MOVL C00497 BC00497 V=1000.0  +MOVJ EC00497 VJ=100.00
'EndPath S3367
'
'Path W3331
SFTOF3D
SFTON3D P053
MOVJ C00498 BC00498 VJ=100.00  +MOVJ EC00498 VJ=100.00
SMOVL C00499 BC00499 V=800.0  +MOVJ EC00499
SMOVL C00500 BC00500 V=150.0 PL=0  +MOVJ EC00500
ARCON
SFTON3D P053
SMOVL C00501 BC00501 V=9.2  +MOVJ EC00501
ARCOF
SMOVL C00502 BC00502 V=800.0  +MOVJ EC00502
SMOVL C00503 BC00503 V=1000.0  +MOVJ EC00503
SFTOF3D
'EndPath W3331
MOVJ C00504 BC00504 VJ=100.00  +MOVJ EC00504 VJ=100.00
'
'Path W3335
SFTOF3D
SFTON3D P051
MOVJ C00505 BC00505 VJ=100.00  +MOVJ EC00505 VJ=100.00
SMOVL C00506 BC00506 V=800.0  +MOVJ EC00506
SMOVL C00507 BC00507 V=150.0 PL=0  +MOVJ EC00507
ARCON
SFTON3D P050
SMOVL C00508 BC00508 V=9.2  +MOVJ EC00508
ARCOF
SMOVL C00509 BC00509 V=800.0  +MOVJ EC00509
SMOVL C00510 BC00510 V=1000.0  +MOVJ EC00510
SFTOF3D
'EndPath W3335
'
'Path W3326
SFTOF3D
SFTON3D P047
MOVJ C00511 BC00511 VJ=100.00  +MOVJ EC00511 VJ=100.00
SMOVL C00512 BC00512 V=800.0  +MOVJ EC00512
SMOVL C00513 BC00513 V=150.0 PL=0  +MOVJ EC00513
MACRO1 MJ#(0) ARGF9
ARCON
SMOVL C00514 BC00514 V=11.7  +MOVJ EC00514
ARCOF
SMOVL C00515 BC00515 V=800.0  +MOVJ EC00515
SMOVL C00516 BC00516 V=1000.0  +MOVJ EC00516
SFTOF3D
'EndPath W3326
'Path W3327
SFTOF3D
SFTON3D P048
MOVJ C00517 BC00517 VJ=100.00  +MOVJ EC00517 VJ=100.00
SMOVL C00518 BC00518 V=800.0  +MOVJ EC00518
SMOVL C00519 BC00519 V=150.0 PL=0  +MOVJ EC00519
ARCON
SMOVL C00520 BC00520 V=11.7  +MOVJ EC00520
ARCOF
SMOVL C00521 BC00521 V=800.0  +MOVJ EC00521
SMOVL C00522 BC00522 V=1000.0  +MOVJ EC00522
SFTOF3D
'EndPath W3327
'Path W3328
SFTOF3D
SFTON3D P049
MOVJ C00523 BC00523 VJ=100.00  +MOVJ EC00523 VJ=100.00
SMOVL C00524 BC00524 V=800.0  +MOVJ EC00524
SMOVL C00525 BC00525 V=150.0 PL=0  +MOVJ EC00525
ARCON
SMOVL C00526 BC00526 V=11.7  +MOVJ EC00526
SMOVL C00527 BC00527 V=11.7  +MOVJ EC00527
ARCOF
SMOVL C00528 BC00528 V=800.0  +MOVJ EC00528
SMOVL C00529 BC00529 V=1000.0  +MOVJ EC00529
SFTOF3D
'EndPath W3328
MOVJ C00530 BC00530 VJ=100.00  +MOVJ EC00530 VJ=100.00
'
'Path W3323
SFTOF3D
SFTON3D P044
MOVJ C00531 BC00531 VJ=100.00  +MOVJ EC00531 VJ=100.00
SMOVL C00532 BC00532 V=800.0  +MOVJ EC00532
SMOVL C00533 BC00533 V=150.0 PL=0  +MOVJ EC00533
ARCON
SMOVL C00534 BC00534 V=11.7  +MOVJ EC00534
SMOVL C00535 BC00535 V=11.7  +MOVJ EC00535
ARCOF
SMOVL C00536 BC00536 V=800.0  +MOVJ EC00536
SMOVL C00537 BC00537 V=1000.0  +MOVJ EC00537
SFTOF3D
'EndPath W3323
'Path W3324
SFTOF3D
SFTON3D P045
MOVJ C00538 BC00538 VJ=100.00  +MOVJ EC00538 VJ=100.00
SMOVL C00539 BC00539 V=800.0  +MOVJ EC00539
SMOVL C00540 BC00540 V=150.0 PL=0  +MOVJ EC00540
ARCON
SMOVL C00541 BC00541 V=11.7  +MOVJ EC00541
ARCOF
SMOVL C00542 BC00542 V=800.0  +MOVJ EC00542
SMOVL C00543 BC00543 V=1000.0  +MOVJ EC00543
SFTOF3D
'EndPath W3324
'Path W3325
SFTOF3D
SFTON3D P046
MOVJ C00544 BC00544 VJ=100.00  +MOVJ EC00544 VJ=100.00
SMOVL C00545 BC00545 V=800.0  +MOVJ EC00545
SMOVL C00546 BC00546 V=150.0 PL=0  +MOVJ EC00546
ARCON
SMOVL C00547 BC00547 V=11.7  +MOVJ EC00547
ARCOF
SMOVL C00548 BC00548 V=800.0  +MOVJ EC00548
SMOVL C00549 BC00549 V=1000.0  +MOVJ EC00549
SFTOF3D
'EndPath W3325
MOVJ C00550 BC00550 VJ=100.00  +MOVJ EC00550 VJ=100.00
'
'
'Path W3320
SFTOF3D
SFTON3D P041
MOVJ C00551 BC00551 VJ=100.00  +MOVJ EC00551 VJ=100.00
SMOVL C00552 BC00552 V=800.0  +MOVJ EC00552
SMOVL C00553 BC00553 V=166.7 PL=0  +MOVJ EC00553
ARCON
SMOVL C00554 BC00554 V=11.7  +MOVJ EC00554
ARCOF
SMOVL C00555 BC00555 V=800.0  +MOVJ EC00555
SMOVL C00556 BC00556 V=1000.0  +MOVJ EC00556
SFTOF3D
'EndPath W3320
'Path W3321
SFTOF3D
SFTON3D P042
MOVJ C00557 BC00557 VJ=100.00  +MOVJ EC00557 VJ=100.00
SMOVL C00558 BC00558 V=800.0  +MOVJ EC00558
SMOVL C00559 BC00559 V=166.7 PL=0  +MOVJ EC00559
ARCON
SMOVL C00560 BC00560 V=11.7  +MOVJ EC00560
ARCOF
SMOVL C00561 BC00561 V=800.0  +MOVJ EC00561
SMOVL C00562 BC00562 V=1000.0  +MOVJ EC00562
SFTOF3D
'EndPath W3321
'Path W3322
SFTOF3D
SFTON3D P043
MOVJ C00563 BC00563 VJ=100.00  +MOVJ EC00563 VJ=100.00
SMOVL C00564 BC00564 V=800.0  +MOVJ EC00564
SMOVL C00565 BC00565 V=166.7 PL=0  +MOVJ EC00565
ARCON
SMOVL C00566 BC00566 V=11.7  +MOVJ EC00566
SMOVL C00567 BC00567 V=11.7  +MOVJ EC00567
ARCOF
SMOVL C00568 BC00568 V=800.0  +MOVJ EC00568
SMOVL C00569 BC00569 V=1000.0  +MOVJ EC00569
SFTOF3D
'EndPath W3322
MOVJ C00570 BC00570 VJ=100.00  +MOVJ EC00570 VJ=100.00
MOVJ C00571 BC00571 VJ=15.00  +MOVJ EC00571 VJ=100.00
MOVJ C00572 BC00572 VJ=15.00  +MOVJ EC00572 VJ=100.00
END
